LIN {X 0,Y 572.959,Z 555.811,A -85,B 0,C 180,E1 -2247.189,E2 -2247.189} C_VEL
LIN {X 0,Y 572.946,Z 558.187,A -85,B 0,C 180,E1 -2248.595,E2 -2248.595} C_VEL
LIN {X 0,Y 572.938,Z 559,A -85,B 0,C 180,E1 -2250.001,E2 -2250.001} C_VEL
LIN {X 0,Y 572.946,Z 558.185,A -85,B 0,C 180,E1 -2251.407,E2 -2251.407} C_VEL
LIN {X 0,Y 572.938,Z 557.198,A -85,B 0,C 180,E1 -2252.11,E2 -2252.11} C_VEL
LIN {X 0,Y 572.959,Z 555.807,A -85,B 0,C 180,E1 -2252.813,E2 -2252.813} C_VEL
LIN {X 0,Y 573.014,Z 552.893,A -85,B 0,C 180,E1 -2253.869,E2 -2253.869} C_VEL
LIN {X 0,Y 572.963,Z 548.945,A -85,B 0,C 180,E1 -2254.927,E2 -2254.927} C_VEL
LIN {X 0,Y 573.068,Z 542.871,A -85,B 0,C 180,E1 -2256.161,E2 -2256.161} C_VEL
LIN {X 0,Y 573.12,Z 536.231,A -85,B 0,C 180,E1 -2257.222,E2 -2257.222} C_VEL
LIN {X 0,Y 573.193,Z 527.983,A -85,B 0,C 180,E1 -2258.284,E2 -2258.284} C_VEL
LIN {X 0,Y 573.32,Z 517.591,A -85,B 0,C 180,E1 -2259.349,E2 -2259.349} C_VEL
LIN {X 0,Y 573.439,Z 507.912,A -85,B 0,C 180,E1 -2260.148,E2 -2260.148} C_VEL
LIN {X 0,Y 573.55,Z 497.389,A -85,B 0,C 180,E1 -2260.855,E2 -2260.855} C_VEL
LIN {X 0,Y 573.651,Z 485.098,A -85,B 0,C 180,E1 -2261.501,E2 -2261.501} C_VEL
LIN {X 0,Y 573.726,Z 473.144,A -85,B 0,C 180,E1 -2261.976,E2 -2261.976} C_VEL
LIN {X 0,Y 573.815,Z 460.48,A -85,B 0,C 180,E1 -2262.333,E2 -2262.333} C_VEL
LIN {X 0,Y 573.91,Z 447.236,A -85,B 0,C 180,E1 -2262.555,E2 -2262.555} C_VEL
LIN {X 0,Y 573.954,Z 350.648,A -85,B 0,C 180,E1 -2263.77,E2 -2263.77} C_VEL
LIN {X 0,Y 573.391,Z 346.606,A -85,B 0,C 180,E1 -2263.852,E2 -2263.852} C_VEL
LIN {X 0,Y 573.57,Z 326.115,A -85,B 0,C 180,E1 -2266.728,E2 -2266.728} C_VEL
LIN {X 0,Y 573.806,Z 305.604,A -85,B 0,C 180,E1 -2269.647,E2 -2269.647} C_VEL
LIN {X 0,Y 574.032,Z 285.767,A -85,B 0,C 180,E1 -2272.496,E2 -2272.496} C_VEL
LIN {X 0,Y 573.584,Z 280.83,A -85,B 0,C 180,E1 -2273.225,E2 -2273.225} C_VEL
LIN {X 0,Y 573.243,Z 279.083,A -85,B 0,C 180,E1 -2273.497,E2 -2273.497} C_VEL
LIN {X 0,Y 573.263,Z 279.079,A -85,B 0,C 180,E1 -2276.191,E2 -2276.191} C_VEL
LIN {X 0,Y 573.238,Z 279.077,A -85,B 0,C 180,E1 -2278.565,E2 -2278.565} C_VEL
LIN {X 0,Y 573.23,Z 279.074,A -85,B 0,C 180,E1 -2280.994,E2 -2280.994} C_VEL
LIN {X 0,Y 573.247,Z 279.073,A -85,B 0,C 180,E1 -2283.521,E2 -2283.521} C_VEL
LIN {X 0,Y 573.219,Z 279.081,A -85,B 0,C 180,E1 -2286.052,E2 -2286.052} C_VEL
LIN {X 0,Y 573.241,Z 279.079,A -85,B 0,C 180,E1 -2288.702,E2 -2288.702} C_VEL
LIN {X 0,Y 573.233,Z 279.074,A -85,B 0,C 180,E1 -2291.593,E2 -2291.593} C_VEL
LIN {X 0,Y 573.227,Z 279.081,A -85,B 0,C 180,E1 -2294.335,E2 -2294.335} C_VEL
LIN {X 0,Y 573.246,Z 279.073,A -85,B 0,C 180,E1 -2297.359,E2 -2297.359} C_VEL
LIN {X 0,Y 573.242,Z 279.077,A -85,B 0,C 180,E1 -2300.392,E2 -2300.392} C_VEL
LIN {X 0,Y 573.257,Z 279.078,A -85,B 0,C 180,E1 -2303.078,E2 -2303.078} C_VEL
LIN {X 0,Y 573.26,Z 279.071,A -85,B 0,C 180,E1 -2305.671,E2 -2305.671} C_VEL
LIN {X 0,Y 573.243,Z 279.073,A -85,B 0,C 180,E1 -2308.184,E2 -2308.184} C_VEL
LIN {X 0,Y 573.268,Z 279.072,A -85,B 0,C 180,E1 -2310.634,E2 -2310.634} C_VEL
LIN {X 0,Y 573.24,Z 279.079,A -85,B 0,C 180,E1 -2313.508,E2 -2313.508} C_VEL
LIN {X 0,Y 573.228,Z 279.075,A -85,B 0,C 180,E1 -2316.134,E2 -2316.134} C_VEL
LIN {X 0,Y 573.255,Z 279.078,A -85,B 0,C 180,E1 -2319.174,E2 -2319.174} C_VEL
LIN {X 0,Y 573.224,Z 279.085,A -85,B 0,C 180,E1 -2321.411,E2 -2321.411} C_VEL
LIN {X 0,Y 573.247,Z 279.082,A -85,B 0,C 180,E1 -2323.621,E2 -2323.621} C_VEL
LIN {X 0,Y 573.276,Z 279.076,A -85,B 0,C 180,E1 -2325.807,E2 -2325.807} C_VEL
LIN {X 0,Y 573.268,Z 279.069,A -85,B 0,C 180,E1 -2328.745,E2 -2328.745} C_VEL
LIN {X 0,Y 573.258,Z 279.077,A -85,B 0,C 180,E1 -2331.54,E2 -2331.54} C_VEL
LIN {X 0,Y 573.29,Z 279.07,A -85,B 0,C 180,E1 -2334.372,E2 -2334.372} C_VEL
LIN {X 0,Y 573.315,Z 279.072,A -85,B 0,C 180,E1 -2337.892,E2 -2337.892} C_VEL
LIN {X 0,Y 573.332,Z 279.063,A -85,B 0,C 180,E1 -2340.702,E2 -2340.702} C_VEL
LIN {X 0,Y 573.234,Z 279.075,A -85,B 0,C 180,E1 -2343.514,E2 -2343.514} C_VEL
LIN {X 0,Y 573.288,Z 279.068,A -85,B 0,C 180,E1 -2345.628,E2 -2345.628} C_VEL
LIN {X 0,Y 573.274,Z 279.07,A -85,B 0,C 180,E1 -2347.75,E2 -2347.75} C_VEL
LIN {X 0,Y 573.267,Z 279.078,A -85,B 0,C 180,E1 -2350.596,E2 -2350.596} C_VEL
LIN {X 0,Y 573.264,Z 279.077,A -85,B 0,C 180,E1 -2352.748,E2 -2352.748} C_VEL
LIN {X 0,Y 573.237,Z 279.079,A -85,B 0,C 180,E1 -2354.92,E2 -2354.92} C_VEL
LIN {X 0,Y 573.242,Z 279.073,A -85,B 0,C 180,E1 -2357.848,E2 -2357.848} C_VEL
LIN {X 0,Y 573.243,Z 279.074,A -85,B 0,C 180,E1 -2360.077,E2 -2360.077} C_VEL
LIN {X 0,Y 573.235,Z 279.076,A -85,B 0,C 180,E1 -2362.338,E2 -2362.338} C_VEL
LIN {X 0,Y 573.25,Z 279.074,A -85,B 0,C 180,E1 -2364.382,E2 -2364.382} C_VEL
LIN {X 0,Y 572.626,Z 279.16,A -85,B 0,C 180,E1 -2364.968,E2 -2364.968} C_VEL
LIN {X 0,Y 569.786,Z 279.516,A -85,B 0,C 180,E1 -2365.92,E2 -2365.92} C_VEL
LIN {X 0,Y 567.352,Z 279.817,A -85,B 0,C 180,E1 -2366.685,E2 -2366.685} C_VEL
LIN {X 0,Y 566.297,Z 279.944,A -85,B 0,C 180,E1 -2367.277,E2 -2367.277} C_VEL
LIN {X 0,Y 566.207,Z 279.952,A -85,B 0,C 180,E1 -2367.477,E2 -2367.477} C_VEL
LIN {X 0,Y 566.205,Z 279.95,A -85,B 0,C 180,E1 -2369.769,E2 -2369.769} C_VEL
LIN {X 0,Y 566.205,Z 279.95,A -85,B 0,C 180,E1 -2372.429,E2 -2372.429} C_VEL
LIN {X 0,Y 566.182,Z 279.958,A -85,B 0,C 180,E1 -2374.989,E2 -2374.989} C_VEL
LIN {X 0,Y 566.195,Z 279.959,A -85,B 0,C 180,E1 -2377.461,E2 -2377.461} C_VEL
LIN {X 0,Y 566.21,Z 279.949,A -85,B 0,C 180,E1 -2380.199,E2 -2380.199} C_VEL
LIN {X 0,Y 566.203,Z 279.953,A -85,B 0,C 180,E1 -2383.054,E2 -2383.054} C_VEL
LIN {X 0,Y 566.197,Z 279.954,A -85,B 0,C 180,E1 -2386.049,E2 -2386.049} C_VEL
LIN {X 0,Y 566.207,Z 279.952,A -85,B 0,C 180,E1 -2389.214,E2 -2389.214} C_VEL
LIN {X 0,Y 566.186,Z 279.96,A -85,B 0,C 180,E1 -2391.636,E2 -2391.636} C_VEL
LIN {X 0,Y 566.165,Z 279.958,A -85,B 0,C 180,E1 -2394.307,E2 -2394.307} C_VEL
LIN {X 0,Y 566.223,Z 279.947,A -85,B 0,C 180,E1 -2396.897,E2 -2396.897} C_VEL
LIN {X 0,Y 566.183,Z 279.953,A -85,B 0,C 180,E1 -2399.407,E2 -2399.407} C_VEL
LIN {X 0,Y 566.215,Z 279.954,A -85,B 0,C 180,E1 -2401.857,E2 -2401.857} C_VEL
LIN {X 0,Y 566.217,Z 279.958,A -85,B 0,C 180,E1 -2404.25,E2 -2404.25} C_VEL
LIN {X 0,Y 566.175,Z 279.957,A -85,B 0,C 180,E1 -2406.718,E2 -2406.718} C_VEL
LIN {X 0,Y 566.215,Z 279.949,A -85,B 0,C 180,E1 -2409.662,E2 -2409.662} C_VEL
LIN {X 0,Y 566.201,Z 279.957,A -85,B 0,C 180,E1 -2412.668,E2 -2412.668} C_VEL
LIN {X 0,Y 566.231,Z 279.946,A -85,B 0,C 180,E1 -2415.626,E2 -2415.626} C_VEL
LIN {X 0,Y 566.237,Z 279.956,A -85,B 0,C 180,E1 -2418.674,E2 -2418.674} C_VEL
LIN {X 0,Y 566.209,Z 279.951,A -85,B 0,C 180,E1 -2421.433,E2 -2421.433} C_VEL
LIN {X 0,Y 566.256,Z 279.947,A -85,B 0,C 180,E1 -2424.301,E2 -2424.301} C_VEL
LIN {X 0,Y 566.218,Z 279.972,A -85,B 0,C 180,E1 -2425.862,E2 -2425.862} C_VEL
LIN {X 0,Y 566.535,Z 283.112,A -85,B 0,C 180,E1 -2426.443,E2 -2426.443} C_VEL
LIN {X 0,Y 566.304,Z 298.68,A -85,B 0,C 180,E1 -2429.288,E2 -2429.288} C_VEL
LIN {X 0,Y 566.19,Z 308.368,A -85,B 0,C 180,E1 -2431.044,E2 -2431.044} C_VEL
LIN {X 0,Y 567.18,Z 314.204,A -85,B 0,C 180,E1 -2431.153,E2 -2431.153} C_VEL
LIN {X 0,Y 566.873,Z 414.703,A -85,B 0,C 180,E1 -2432.441,E2 -2432.441} C_VEL
LIN {X 0,Y 566.763,Z 427.913,A -85,B 0,C 180,E1 -2432.753,E2 -2432.753} C_VEL
LIN {X 0,Y 566.723,Z 440.499,A -85,B 0,C 180,E1 -2433.198,E2 -2433.198} C_VEL
LIN {X 0,Y 566.588,Z 451.79,A -85,B 0,C 180,E1 -2433.733,E2 -2433.733} C_VEL
LIN {X 0,Y 566.408,Z 463.445,A -85,B 0,C 180,E1 -2434.447,E2 -2434.447} C_VEL
LIN {X 0,Y 566.309,Z 473.897,A -85,B 0,C 180,E1 -2435.25,E2 -2435.25} C_VEL
LIN {X 0,Y 566.171,Z 482.489,A -85,B 0,C 180,E1 -2436.056,E2 -2436.056} C_VEL
LIN {X 0,Y 566.111,Z 490.229,A -85,B 0,C 180,E1 -2436.928,E2 -2436.928} C_VEL
LIN {X 0,Y 566.043,Z 498.223,A -85,B 0,C 180,E1 -2438.028,E2 -2438.028} C_VEL
LIN {X 0,Y 565.981,Z 503.555,A -85,B 0,C 180,E1 -2438.928,E2 -2438.928} C_VEL
LIN {X 0,Y 565.946,Z 508.754,A -85,B 0,C 180,E1 -2440.011,E2 -2440.011} C_VEL
LIN {X 0,Y 565.929,Z 513.016,A -85,B 0,C 180,E1 -2441.169,E2 -2441.169} C_VEL
LIN {X 0,Y 565.867,Z 515.788,A -85,B 0,C 180,E1 -2442.188,E2 -2442.188} C_VEL
LIN {X 0,Y 565.843,Z 517.211,A -85,B 0,C 180,E1 -2442.917,E2 -2442.917} C_VEL
LIN {X 0,Y 565.861,Z 518.215,A -85,B 0,C 180,E1 -2443.648,E2 -2443.648} C_VEL
LIN {X 0,Y 565.873,Z 518.817,A -85,B 0,C 180,E1 -2444.381,E2 -2444.381} C_VEL
LIN {X 0,Y 565.803,Z 518.99,A -85,B 0,C 180,E1 -2445.119,E2 -2445.119} C_VEL
LIN {X 0,Y 565.81,Z 518.719,A -85,B 0,C 180,E1 -2445.857,E2 -2445.857} C_VEL
LIN {X 0,Y 565.851,Z 517.497,A -85,B 0,C 180,E1 -2446.99,E2 -2446.99} C_VEL
LIN {X 0,Y 565.892,Z 514.38,A -85,B 0,C 180,E1 -2448.462,E2 -2448.462} C_VEL
LIN {X 0,Y 565.926,Z 510.712,A -85,B 0,C 180,E1 -2449.59,E2 -2449.59} C_VEL
LIN {X 0,Y 565.944,Z 505.785,A -85,B 0,C 180,E1 -2450.726,E2 -2450.726} C_VEL
LIN {X 0,Y 566.004,Z 499.43,A -85,B 0,C 180,E1 -2451.869,E2 -2451.869} C_VEL
LIN {X 0,Y 566.077,Z 491.551,A -85,B 0,C 180,E1 -2452.998,E2 -2452.998} C_VEL
LIN {X 0,Y 566.184,Z 482.955,A -85,B 0,C 180,E1 -2453.985,E2 -2453.985} C_VEL
LIN {X 0,Y 566.315,Z 473.683,A -85,B 0,C 180,E1 -2454.858,E2 -2454.858} C_VEL
LIN {X 0,Y 566.454,Z 463.473,A -85,B 0,C 180,E1 -2455.64,E2 -2455.64} C_VEL
LIN {X 0,Y 566.6,Z 452.432,A -85,B 0,C 180,E1 -2456.322,E2 -2456.322} C_VEL
LIN {X 0,Y 566.745,Z 440.606,A -85,B 0,C 180,E1 -2456.888,E2 -2456.888} C_VEL
LIN {X 0,Y 566.832,Z 428.098,A -85,B 0,C 180,E1 -2457.33,E2 -2457.33} C_VEL
LIN {X 0,Y 566.919,Z 414.525,A -85,B 0,C 180,E1 -2457.651,E2 -2457.651} C_VEL
LIN {X 0,Y 567.043,Z 313.459,A -85,B 0,C 180,E1 -2458.95,E2 -2458.95} C_VEL
LIN {X 0,Y 566.206,Z 308.331,A -85,B 0,C 180,E1 -2459.053,E2 -2459.053} C_VEL
LIN {X 0,Y 566.364,Z 293.061,A -85,B 0,C 180,E1 -2461.827,E2 -2461.827} C_VEL
LIN {X 0,Y 566.379,Z 281.442,A -85,B 0,C 180,E1 -2463.943,E2 -2463.943} C_VEL
LIN {X 0,Y 566.14,Z 279.963,A -85,B 0,C 180,E1 -2464.227,E2 -2464.227} C_VEL
LIN {X 0,Y 566.176,Z 279.962,A -85,B 0,C 180,E1 -2467.461,E2 -2467.461} C_VEL
LIN {X 0,Y 566.181,Z 279.954,A -85,B 0,C 180,E1 -2470.199,E2 -2470.199} C_VEL
LIN {X 0,Y 566.13,Z 279.965,A -85,B 0,C 180,E1 -2473.059,E2 -2473.059} C_VEL
LIN {X 0,Y 566.143,Z 279.958,A -85,B 0,C 180,E1 -2476.052,E2 -2476.052} C_VEL
LIN {X 0,Y 566.142,Z 279.959,A -85,B 0,C 180,E1 -2478.858,E2 -2478.858} C_VEL
LIN {X 0,Y 566.186,Z 279.961,A -85,B 0,C 180,E1 -2481.442,E2 -2481.442} C_VEL
LIN {X 0,Y 566.125,Z 279.958,A -85,B 0,C 180,E1 -2484.305,E2 -2484.305} C_VEL
LIN {X 0,Y 566.189,Z 279.953,A -85,B 0,C 180,E1 -2486.896,E2 -2486.896} C_VEL
LIN {X 0,Y 566.162,Z 279.959,A -85,B 0,C 180,E1 -2489.406,E2 -2489.406} C_VEL
LIN {X 0,Y 566.172,Z 279.964,A -85,B 0,C 180,E1 -2491.855,E2 -2491.855} C_VEL
LIN {X 0,Y 566.222,Z 279.947,A -85,B 0,C 180,E1 -2495.039,E2 -2495.039} C_VEL
LIN {X 0,Y 566.176,Z 279.96,A -85,B 0,C 180,E1 -2498.137,E2 -2498.137} C_VEL
LIN {X 0,Y 566.215,Z 279.951,A -85,B 0,C 180,E1 -2500.613,E2 -2500.613} C_VEL
LIN {X 0,Y 566.163,Z 279.955,A -85,B 0,C 180,E1 -2503.411,E2 -2503.411} C_VEL
LIN {X 0,Y 566.174,Z 279.96,A -85,B 0,C 180,E1 -2506.358,E2 -2506.358} C_VEL
LIN {X 0,Y 566.219,Z 279.951,A -85,B 0,C 180,E1 -2508.675,E2 -2508.675} C_VEL
LIN {X 0,Y 566.21,Z 279.949,A -85,B 0,C 180,E1 -2511.434,E2 -2511.434} C_VEL
LIN {X 0,Y 566.243,Z 279.953,A -85,B 0,C 180,E1 -2514.302,E2 -2514.302} C_VEL
LIN {X 0,Y 566.256,Z 279.944,A -85,B 0,C 180,E1 -2517.866,E2 -2517.866} C_VEL
LIN {X 0,Y 566.297,Z 279.945,A -85,B 0,C 180,E1 -2520.711,E2 -2520.711} C_VEL
LIN {X 0,Y 566.173,Z 279.952,A -85,B 0,C 180,E1 -2523.559,E2 -2523.559} C_VEL
LIN {X 0,Y 566.243,Z 279.945,A -85,B 0,C 180,E1 -2525.699,E2 -2525.699} C_VEL
LIN {X 0,Y 566.22,Z 279.955,A -85,B 0,C 180,E1 -2528.566,E2 -2528.566} C_VEL
LIN {X 0,Y 566.237,Z 279.947,A -85,B 0,C 180,E1 -2531.455,E2 -2531.455} C_VEL
LIN {X 0,Y 566.22,Z 279.951,A -85,B 0,C 180,E1 -2534.507,E2 -2534.507} C_VEL
LIN {X 0,Y 566.186,Z 279.955,A -85,B 0,C 180,E1 -2537.332,E2 -2537.332} C_VEL
LIN {X 0,Y 566.2,Z 279.951,A -85,B 0,C 180,E1 -2540.338,E2 -2540.338} C_VEL
LIN {X 0,Y 566.177,Z 279.957,A -85,B 0,C 180,E1 -2543.405,E2 -2543.405} C_VEL
LIN {X 0,Y 566.215,Z 279.95,A -85,B 0,C 180,E1 -2545.749,E2 -2545.749} C_VEL
LIN {X 0,Y 566.19,Z 279.95,A -85,B 0,C 180,E1 -2548.203,E2 -2548.203} C_VEL
LIN {X 0,Y 566.183,Z 279.954,A -85,B 0,C 180,E1 -2550.593,E2 -2550.593} C_VEL
LIN {X 0,Y 566.218,Z 279.954,A -85,B 0,C 180,E1 -2553.103,E2 -2553.103} C_VEL
LIN {X 0,Y 566.202,Z 279.955,A -85,B 0,C 180,E1 -2555.69,E2 -2555.69} C_VEL
LIN {X 0,Y 566.207,Z 279.95,A -85,B 0,C 180,E1 -2558.56,E2 -2558.56} C_VEL
LIN {X 0,Y 566.203,Z 279.955,A -85,B 0,C 180,E1 -2561.137,E2 -2561.137} C_VEL
LIN {X 0,Y 566.192,Z 279.954,A -85,B 0,C 180,E1 -2564.037,E2 -2564.037} C_VEL
LIN {X 0,Y 566.198,Z 279.952,A -85,B 0,C 180,E1 -2567.084,E2 -2567.084} C_VEL
LIN {X 0,Y 566.22,Z 279.956,A -85,B 0,C 180,E1 -2569.804,E2 -2569.804} C_VEL
LIN {X 0,Y 566.194,Z 279.952,A -85,B 0,C 180,E1 -2572.6,E2 -2572.6} C_VEL
LIN {X 0,Y 566.204,Z 279.952,A -85,B 0,C 180,E1 -2575.184,E2 -2575.184} C_VEL
LIN {X 0,Y 566.226,Z 279.956,A -85,B 0,C 180,E1 -2577.745,E2 -2577.745} C_VEL
LIN {X 0,Y 566.2,Z 279.956,A -85,B 0,C 180,E1 -2580.329,E2 -2580.329} C_VEL
LIN {X 0,Y 566.216,Z 279.951,A -85,B 0,C 180,E1 -2582.663,E2 -2582.663} C_VEL
LIN {X 0,Y 566.234,Z 279.949,A -85,B 0,C 180,E1 -2585.04,E2 -2585.04} C_VEL
LIN {X 0,Y 566.222,Z 280.105,A -85,B 0,C 180,E1 -2586.405,E2 -2586.405} C_VEL
LIN {X 0,Y 567.058,Z 285.451,A -85,B 0,C 180,E1 -2587.214,E2 -2587.214} C_VEL
LIN {X 0,Y 566.867,Z 306.727,A -85,B 0,C 180,E1 -2590.275,E2 -2590.275} C_VEL
LIN {X 0,Y 566.598,Z 327.558,A -85,B 0,C 180,E1 -2593.267,E2 -2593.267} C_VEL
LIN {X 0,Y 566.392,Z 346.703,A -85,B 0,C 180,E1 -2595.987,E2 -2595.987} C_VEL
LIN {X 0,Y 567.202,Z 353.339,A -85,B 0,C 180,E1 -2596.097,E2 -2596.097} C_VEL
LIN {X 0,Y 566.952,Z 455.008,A -85,B 0,C 180,E1 -2597.404,E2 -2597.404} C_VEL
LIN {X 0,Y 566.836,Z 468.259,A -85,B 0,C 180,E1 -2597.72,E2 -2597.72} C_VEL
LIN {X 0,Y 566.719,Z 480.407,A -85,B 0,C 180,E1 -2598.149,E2 -2598.149} C_VEL
LIN {X 0,Y 566.626,Z 492.089,A -85,B 0,C 180,E1 -2598.705,E2 -2598.705} C_VEL
LIN {X 0,Y 566.487,Z 502.924,A -85,B 0,C 180,E1 -2599.367,E2 -2599.367} C_VEL
LIN {X 0,Y 566.329,Z 513.554,A -85,B 0,C 180,E1 -2600.177,E2 -2600.177} C_VEL
LIN {X 0,Y 566.205,Z 523.094,A -85,B 0,C 180,E1 -2601.075,E2 -2601.075} C_VEL
LIN {X 0,Y 566.11,Z 530.97,A -85,B 0,C 180,E1 -2601.973,E2 -2601.973} C_VEL
LIN {X 0,Y 566.004,Z 538.629,A -85,B 0,C 180,E1 -2603.048,E2 -2603.048} C_VEL
LIN {X 0,Y 566.004,Z 545.685,A -85,B 0,C 180,E1 -2604.3,E2 -2604.3} C_VEL
LIN {X 0,Y 565.933,Z 550.377,A -85,B 0,C 180,E1 -2605.371,E2 -2605.371} C_VEL
LIN {X 0,Y 565.926,Z 553.961,A -85,B 0,C 180,E1 -2606.441,E2 -2606.441} C_VEL
LIN {X 0,Y 565.877,Z 555.81,A -85,B 0,C 180,E1 -2607.154,E2 -2607.154} C_VEL
LIN {X 0,Y 565.845,Z 558.186,A -85,B 0,C 180,E1 -2608.578,E2 -2608.578} C_VEL
LIN {X 0,Y 565.839,Z 559,A -85,B 0,C 180,E1 -2610.001,E2 -2610.001} C_VEL
LIN {X 0,Y 565.845,Z 558.184,A -85,B 0,C 180,E1 -2611.424,E2 -2611.424} C_VEL
LIN {X 0,Y 565.878,Z 555.808,A -85,B 0,C 180,E1 -2612.849,E2 -2612.849} C_VEL
LIN {X 0,Y 565.926,Z 552.893,A -85,B 0,C 180,E1 -2613.917,E2 -2613.917} C_VEL
LIN {X 0,Y 565.878,Z 548.945,A -85,B 0,C 180,E1 -2614.988,E2 -2614.988} C_VEL
LIN {X 0,Y 565.994,Z 542.871,A -85,B 0,C 180,E1 -2616.238,E2 -2616.238} C_VEL
LIN {X 0,Y 566.053,Z 536.23,A -85,B 0,C 180,E1 -2617.312,E2 -2617.312} C_VEL
LIN {X 0,Y 566.142,Z 527.983,A -85,B 0,C 180,E1 -2618.388,E2 -2618.388} C_VEL
LIN {X 0,Y 566.254,Z 519.529,A -85,B 0,C 180,E1 -2619.286,E2 -2619.286} C_VEL
LIN {X 0,Y 566.393,Z 509.083,A -85,B 0,C 180,E1 -2620.185,E2 -2620.185} C_VEL
LIN {X 0,Y 566.571,Z 497.689,A -85,B 0,C 180,E1 -2620.972,E2 -2620.972} C_VEL
LIN {X 0,Y 566.693,Z 485.866,A -85,B 0,C 180,E1 -2621.609,E2 -2621.609} C_VEL
LIN {X 0,Y 566.777,Z 473.142,A -85,B 0,C 180,E1 -2622.125,E2 -2622.125} C_VEL
LIN {X 0,Y 566.878,Z 460.479,A -85,B 0,C 180,E1 -2622.486,E2 -2622.486} C_VEL
LIN {X 0,Y 566.978,Z 447.236,A -85,B 0,C 180,E1 -2622.711,E2 -2622.711} C_VEL
LIN {X 0,Y 567.048,Z 351.206,A -85,B 0,C 180,E1 -2623.934,E2 -2623.934} C_VEL
LIN {X 0,Y 566.385,Z 346.606,A -85,B 0,C 180,E1 -2624.026,E2 -2624.026} C_VEL
LIN {X 0,Y 566.613,Z 324.886,A -85,B 0,C 180,E1 -2627.116,E2 -2627.116} C_VEL
LIN {X 0,Y 566.87,Z 303.955,A -85,B 0,C 180,E1 -2630.124,E2 -2630.124} C_VEL
LIN {X 0,Y 567.057,Z 285.517,A -85,B 0,C 180,E1 -2632.788,E2 -2632.788} C_VEL
LIN {X 0,Y 566.21,Z 279.959,A -85,B 0,C 180,E1 -2633.646,E2 -2633.646} C_VEL
LIN {X 0,Y 566.212,Z 279.958,A -85,B 0,C 180,E1 -2635.75,E2 -2635.75} C_VEL
LIN {X 0,Y 566.209,Z 279.958,A -85,B 0,C 180,E1 -2638.203,E2 -2638.203} C_VEL
LIN {X 0,Y 566.195,Z 279.951,A -85,B 0,C 180,E1 -2641.077,E2 -2641.077} C_VEL
LIN {X 0,Y 566.203,Z 279.952,A -85,B 0,C 180,E1 -2643.732,E2 -2643.732} C_VEL
LIN {X 0,Y 566.205,Z 279.956,A -85,B 0,C 180,E1 -2646.57,E2 -2646.57} C_VEL
LIN {X 0,Y 566.217,Z 279.948,A -85,B 0,C 180,E1 -2649.686,E2 -2649.686} C_VEL
LIN {X 0,Y 566.206,Z 279.954,A -85,B 0,C 180,E1 -2652.917,E2 -2652.917} C_VEL
LIN {X 0,Y 566.199,Z 279.952,A -85,B 0,C 180,E1 -2656.049,E2 -2656.049} C_VEL
LIN {X 0,Y 566.209,Z 279.952,A -85,B 0,C 180,E1 -2659.215,E2 -2659.215} C_VEL
LIN {X 0,Y 566.188,Z 279.952,A -85,B 0,C 180,E1 -2661.637,E2 -2661.637} C_VEL
LIN {X 0,Y 566.167,Z 279.956,A -85,B 0,C 180,E1 -2664.308,E2 -2664.308} C_VEL
LIN {X 0,Y 566.205,Z 279.958,A -85,B 0,C 180,E1 -2666.897,E2 -2666.897} C_VEL
LIN {X 0,Y 566.185,Z 279.957,A -85,B 0,C 180,E1 -2669.407,E2 -2669.407} C_VEL
LIN {X 0,Y 566.199,Z 279.951,A -85,B 0,C 180,E1 -2671.856,E2 -2671.856} C_VEL
LIN {X 0,Y 566.213,Z 279.948,A -85,B 0,C 180,E1 -2674.251,E2 -2674.251} C_VEL
LIN {X 0,Y 566.173,Z 279.955,A -85,B 0,C 180,E1 -2676.72,E2 -2676.72} C_VEL
LIN {X 0,Y 566.212,Z 279.955,A -85,B 0,C 180,E1 -2679.663,E2 -2679.663} C_VEL
LIN {X 0,Y 566.199,Z 279.95,A -85,B 0,C 180,E1 -2682.668,E2 -2682.668} C_VEL
LIN {X 0,Y 566.238,Z 279.956,A -85,B 0,C 180,E1 -2685.627,E2 -2685.627} C_VEL
LIN {X 0,Y 566.24,Z 279.945,A -85,B 0,C 180,E1 -2688.675,E2 -2688.675} C_VEL
LIN {X 0,Y 566.209,Z 279.953,A -85,B 0,C 180,E1 -2691.434,E2 -2691.434} C_VEL
LIN {X 0,Y 566.256,Z 279.947,A -85,B 0,C 180,E1 -2694.302,E2 -2694.302} C_VEL
LIN {X 0,Y 566.286,Z 279.947,A -85,B 0,C 180,E1 -2697.866,E2 -2697.866} C_VEL
LIN {X 0,Y 566.303,Z 279.939,A -85,B 0,C 180,E1 -2700.711,E2 -2700.711} C_VEL
LIN {X 0,Y 566.273,Z 279.942,A -85,B 0,C 180,E1 -2702.845,E2 -2702.845} C_VEL
LIN {X 0,Y 566.256,Z 279.945,A -85,B 0,C 180,E1 -2705.698,E2 -2705.698} C_VEL
LIN {X 0,Y 566.209,Z 279.956,A -85,B 0,C 180,E1 -2708.566,E2 -2708.566} C_VEL
LIN {X 0,Y 566.247,Z 279.944,A -85,B 0,C 180,E1 -2711.454,E2 -2711.454} C_VEL
LIN {X 0,Y 566.234,Z 279.955,A -85,B 0,C 180,E1 -2714.504,E2 -2714.504} C_VEL
LIN {X 0,Y 566.201,Z 279.951,A -85,B 0,C 180,E1 -2717.331,E2 -2717.331} C_VEL
LIN {X 0,Y 566.21,Z 279.952,A -85,B 0,C 180,E1 -2720.337,E2 -2720.337} C_VEL
LIN {X 0,Y 566.172,Z 279.957,A -85,B 0,C 180,E1 -2723.28,E2 -2723.28} C_VEL
LIN {X 0,Y 566.217,Z 279.948,A -85,B 0,C 180,E1 -2725.749,E2 -2725.749} C_VEL
LIN {X 0,Y 566.207,Z 279.952,A -85,B 0,C 180,E1 -2727.477,E2 -2727.477} C_VEL
LIN {X 0,Y 565.527,Z 280.037,A -85,B 0,C 180,E1 -2728.071,E2 -2728.071} C_VEL
LIN {X 0,Y 562.661,Z 280.402,A -85,B 0,C 180,E1 -2729.034,E2 -2729.034} C_VEL
LIN {X 0,Y 560.251,Z 280.696,A -85,B 0,C 180,E1 -2729.81,E2 -2729.81} C_VEL
LIN {X 0,Y 559.223,Z 280.82,A -85,B 0,C 180,E1 -2730.408,E2 -2730.408} C_VEL
LIN {X 0,Y 559.143,Z 280.832,A -85,B 0,C 180,E1 -2730.611,E2 -2730.611} C_VEL
LIN {X 0,Y 559.166,Z 280.831,A -85,B 0,C 180,E1 -2733.575,E2 -2733.575} C_VEL
LIN {X 0,Y 559.133,Z 280.831,A -85,B 0,C 180,E1 -2736.442,E2 -2736.442} C_VEL
LIN {X 0,Y 559.176,Z 280.828,A -85,B 0,C 180,E1 -2738.934,E2 -2738.934} C_VEL
LIN {X 0,Y 559.167,Z 280.832,A -85,B 0,C 180,E1 -2741.77,E2 -2741.77} C_VEL
LIN {X 0,Y 559.135,Z 280.83,A -85,B 0,C 180,E1 -2744.74,E2 -2744.74} C_VEL
LIN {X 0,Y 559.161,Z 280.831,A -85,B 0,C 180,E1 -2747.256,E2 -2747.256} C_VEL
LIN {X 0,Y 559.181,Z 280.829,A -85,B 0,C 180,E1 -2750.134,E2 -2750.134} C_VEL
LIN {X 0,Y 559.144,Z 280.829,A -85,B 0,C 180,E1 -2752.891,E2 -2752.891} C_VEL
LIN {X 0,Y 559.169,Z 280.835,A -85,B 0,C 180,E1 -2756.05,E2 -2756.05} C_VEL
LIN {X 0,Y 559.157,Z 280.827,A -85,B 0,C 180,E1 -2758.98,E2 -2758.98} C_VEL
LIN {X 0,Y 559.172,Z 280.828,A -85,B 0,C 180,E1 -2761.618,E2 -2761.618} C_VEL
LIN {X 0,Y 559.184,Z 280.829,A -85,B 0,C 180,E1 -2763.902,E2 -2763.902} C_VEL
LIN {X 0,Y 559.145,Z 280.835,A -85,B 0,C 180,E1 -2766.57,E2 -2766.57} C_VEL
LIN {X 0,Y 559.182,Z 280.824,A -85,B 0,C 180,E1 -2769.395,E2 -2769.395} C_VEL
LIN {X 0,Y 559.143,Z 280.83,A -85,B 0,C 180,E1 -2771.685,E2 -2771.685} C_VEL
LIN {X 0,Y 559.166,Z 280.828,A -85,B 0,C 180,E1 -2773.947,E2 -2773.947} C_VEL
LIN {X 0,Y 559.17,Z 280.829,A -85,B 0,C 180,E1 -2776.183,E2 -2776.183} C_VEL
LIN {X 0,Y 559.208,Z 280.83,A -85,B 0,C 180,E1 -2778.604,E2 -2778.604} C_VEL
LIN {X 0,Y 559.173,Z 280.829,A -85,B 0,C 180,E1 -2781.324,E2 -2781.324} C_VEL
LIN {X 0,Y 559.225,Z 280.823,A -85,B 0,C 180,E1 -2784.229,E2 -2784.229} C_VEL
LIN {X 0,Y 559.18,Z 280.84,A -85,B 0,C 180,E1 -2785.81,E2 -2785.81} C_VEL
LIN {X 0,Y 559.473,Z 285.017,A -85,B 0,C 180,E1 -2786.578,E2 -2786.578} C_VEL
LIN {X 0,Y 559.277,Z 299.735,A -85,B 0,C 180,E1 -2789.279,E2 -2789.279} C_VEL
LIN {X 0,Y 559.173,Z 308.573,A -85,B 0,C 180,E1 -2790.877,E2 -2790.877} C_VEL
LIN {X 0,Y 560.267,Z 314.934,A -85,B 0,C 180,E1 -2790.987,E2 -2790.987} C_VEL
LIN {X 0,Y 559.941,Z 415.154,A -85,B 0,C 180,E1 -2792.292,E2 -2792.292} C_VEL
LIN {X 0,Y 559.827,Z 428.204,A -85,B 0,C 180,E1 -2792.607,E2 -2792.607} C_VEL
LIN {X 0,Y 559.776,Z 440.715,A -85,B 0,C 180,E1 -2793.058,E2 -2793.058} C_VEL
LIN {X 0,Y 559.619,Z 451.958,A -85,B 0,C 180,E1 -2793.599,E2 -2793.599} C_VEL
LIN {X 0,Y 559.408,Z 463.576,A -85,B 0,C 180,E1 -2794.322,E2 -2794.322} C_VEL
LIN {X 0,Y 559.31,Z 474,A -85,B 0,C 180,E1 -2795.135,E2 -2795.135} C_VEL
LIN {X 0,Y 559.12,Z 482.587,A -85,B 0,C 180,E1 -2795.951,E2 -2795.951} C_VEL
LIN {X 0,Y 559.069,Z 490.681,A -85,B 0,C 180,E1 -2796.88,E2 -2796.88} C_VEL
LIN {X 0,Y 558.98,Z 498.281,A -85,B 0,C 180,E1 -2797.948,E2 -2797.948} C_VEL
LIN {X 0,Y 558.877,Z 504.538,A -85,B 0,C 180,E1 -2799.043,E2 -2799.043} C_VEL
LIN {X 0,Y 558.852,Z 509.517,A -85,B 0,C 180,E1 -2800.139,E2 -2800.139} C_VEL
LIN {X 0,Y 558.844,Z 513.281,A -85,B 0,C 180,E1 -2801.209,E2 -2801.209} C_VEL
LIN {X 0,Y 558.772,Z 516.187,A -85,B 0,C 180,E1 -2802.345,E2 -2802.345} C_VEL
LIN {X 0,Y 558.742,Z 517.512,A -85,B 0,C 180,E1 -2803.084,E2 -2803.084} C_VEL
LIN {X 0,Y 558.786,Z 518.854,A -85,B 0,C 180,E1 -2804.431,E2 -2804.431} C_VEL
LIN {X 0,Y 558.706,Z 518.947,A -85,B 0,C 180,E1 -2805.316,E2 -2805.316} C_VEL
LIN {X 0,Y 558.727,Z 518.588,A -85,B 0,C 180,E1 -2806.064,E2 -2806.064} C_VEL
LIN {X 0,Y 558.76,Z 517.4,A -85,B 0,C 180,E1 -2807.076,E2 -2807.076} C_VEL
LIN {X 0,Y 558.777,Z 514.835,A -85,B 0,C 180,E1 -2808.325,E2 -2808.325} C_VEL
LIN {X 0,Y 558.826,Z 511.585,A -85,B 0,C 180,E1 -2809.399,E2 -2809.399} C_VEL
LIN {X 0,Y 558.841,Z 506.657,A -85,B 0,C 180,E1 -2810.616,E2 -2810.616} C_VEL
LIN {X 0,Y 558.913,Z 500.718,A -85,B 0,C 180,E1 -2811.746,E2 -2811.746} C_VEL
LIN {X 0,Y 559.001,Z 492.76,A -85,B 0,C 180,E1 -2812.937,E2 -2812.937} C_VEL
LIN {X 0,Y 559.134,Z 484.696,A -85,B 0,C 180,E1 -2813.912,E2 -2813.912} C_VEL
LIN {X 0,Y 559.292,Z 474.717,A -85,B 0,C 180,E1 -2814.894,E2 -2814.894} C_VEL
LIN {X 0,Y 559.458,Z 463.372,A -85,B 0,C 180,E1 -2815.782,E2 -2815.782} C_VEL
LIN {X 0,Y 559.629,Z 452.253,A -85,B 0,C 180,E1 -2816.474,E2 -2816.474} C_VEL
LIN {X 0,Y 559.806,Z 440.738,A -85,B 0,C 180,E1 -2817.031,E2 -2817.031} C_VEL
LIN {X 0,Y 559.898,Z 428.358,A -85,B 0,C 180,E1 -2817.477,E2 -2817.477} C_VEL
LIN {X 0,Y 559.982,Z 415.296,A -85,B 0,C 180,E1 -2817.794,E2 -2817.794} C_VEL
LIN {X 0,Y 560.224,Z 314.878,A -85,B 0,C 180,E1 -2819.105,E2 -2819.105} C_VEL
LIN {X 0,Y 559.186,Z 308.391,A -85,B 0,C 180,E1 -2819.221,E2 -2819.221} C_VEL
LIN {X 0,Y 559.346,Z 292.939,A -85,B 0,C 180,E1 -2822.054,E2 -2822.054} C_VEL
LIN {X 0,Y 559.328,Z 282.22,A -85,B 0,C 180,E1 -2823.974,E2 -2823.974} C_VEL
LIN {X 0,Y 559.104,Z 280.84,A -85,B 0,C 180,E1 -2824.25,E2 -2824.25} C_VEL
LIN {X 0,Y 559.105,Z 280.844,A -85,B 0,C 180,E1 -2827.109,E2 -2827.109} C_VEL
LIN {X 0,Y 559.133,Z 280.833,A -85,B 0,C 180,E1 -2829.938,E2 -2829.938} C_VEL
LIN {X 0,Y 559.097,Z 280.838,A -85,B 0,C 180,E1 -2832.747,E2 -2832.747} C_VEL
LIN {X 0,Y 559.109,Z 280.838,A -85,B 0,C 180,E1 -2835.763,E2 -2835.763} C_VEL
LIN {X 0,Y 559.111,Z 280.835,A -85,B 0,C 180,E1 -2838.225,E2 -2838.225} C_VEL
LIN {X 0,Y 559.154,Z 280.833,A -85,B 0,C 180,E1 -2841.192,E2 -2841.192} C_VEL
LIN {X 0,Y 559.1,Z 280.839,A -85,B 0,C 180,E1 -2843.786,E2 -2843.786} C_VEL
LIN {X 0,Y 559.133,Z 280.832,A -85,B 0,C 180,E1 -2846.423,E2 -2846.423} C_VEL
LIN {X 0,Y 559.138,Z 280.83,A -85,B 0,C 180,E1 -2848.98,E2 -2848.98} C_VEL
LIN {X 0,Y 559.119,Z 280.84,A -85,B 0,C 180,E1 -2851.625,E2 -2851.625} C_VEL
LIN {X 0,Y 559.164,Z 280.826,A -85,B 0,C 180,E1 -2854.813,E2 -2854.813} C_VEL
LIN {X 0,Y 559.124,Z 280.841,A -85,B 0,C 180,E1 -2857.847,E2 -2857.847} C_VEL
LIN {X 0,Y 559.176,Z 280.829,A -85,B 0,C 180,E1 -2860.494,E2 -2860.494} C_VEL
LIN {X 0,Y 559.141,Z 280.828,A -85,B 0,C 180,E1 -2863.196,E2 -2863.196} C_VEL
LIN {X 0,Y 559.148,Z 280.839,A -85,B 0,C 180,E1 -2866.184,E2 -2866.184} C_VEL
LIN {X 0,Y 559.19,Z 280.827,A -85,B 0,C 180,E1 -2868.605,E2 -2868.605} C_VEL
LIN {X 0,Y 559.169,Z 280.826,A -85,B 0,C 180,E1 -2871.325,E2 -2871.325} C_VEL
LIN {X 0,Y 559.21,Z 280.828,A -85,B 0,C 180,E1 -2874.23,E2 -2874.23} C_VEL
LIN {X 0,Y 559.228,Z 280.819,A -85,B 0,C 180,E1 -2877.839,E2 -2877.839} C_VEL
LIN {X 0,Y 559.266,Z 280.821,A -85,B 0,C 180,E1 -2880.72,E2 -2880.72} C_VEL
LIN {X 0,Y 559.234,Z 280.821,A -85,B 0,C 180,E1 -2882.882,E2 -2882.882} C_VEL
LIN {X 0,Y 559.212,Z 280.821,A -85,B 0,C 180,E1 -2885.771,E2 -2885.771} C_VEL
LIN {X 0,Y 559.179,Z 280.833,A -85,B 0,C 180,E1 -2888.675,E2 -2888.675} C_VEL
LIN {X 0,Y 559.195,Z 280.823,A -85,B 0,C 180,E1 -2891.601,E2 -2891.601} C_VEL
LIN {X 0,Y 559.186,Z 280.828,A -85,B 0,C 180,E1 -2894.596,E2 -2894.596} C_VEL
LIN {X 0,Y 559.146,Z 280.83,A -85,B 0,C 180,E1 -2897.558,E2 -2897.558} C_VEL
LIN {X 0,Y 559.159,Z 280.827,A -85,B 0,C 180,E1 -2899.838,E2 -2899.838} C_VEL
LIN {X 0,Y 559.128,Z 280.831,A -85,B 0,C 180,E1 -2902.154,E2 -2902.154} C_VEL
LIN {X 0,Y 559.167,Z 280.836,A -85,B 0,C 180,E1 -2905.188,E2 -2905.188} C_VEL
LIN {X 0,Y 559.181,Z 280.825,A -85,B 0,C 180,E1 -2907.712,E2 -2907.712} C_VEL
LIN {X 0,Y 559.158,Z 280.828,A -85,B 0,C 180,E1 -2910.183,E2 -2910.183} C_VEL
LIN {X 0,Y 559.165,Z 280.828,A -85,B 0,C 180,E1 -2912.715,E2 -2912.715} C_VEL
LIN {X 0,Y 559.147,Z 280.839,A -85,B 0,C 180,E1 -2915.323,E2 -2915.323} C_VEL
LIN {X 0,Y 559.126,Z 280.834,A -85,B 0,C 180,E1 -2918.018,E2 -2918.018} C_VEL
LIN {X 0,Y 559.168,Z 280.828,A -85,B 0,C 180,E1 -2920.812,E2 -2920.812} C_VEL
LIN {X 0,Y 559.154,Z 280.835,A -85,B 0,C 180,E1 -2923.733,E2 -2923.733} C_VEL
LIN {X 0,Y 559.161,Z 280.826,A -85,B 0,C 180,E1 -2926.802,E2 -2926.802} C_VEL
LIN {X 0,Y 559.17,Z 280.829,A -85,B 0,C 180,E1 -2929.191,E2 -2929.191} C_VEL
LIN {X 0,Y 559.129,Z 280.838,A -85,B 0,C 180,E1 -2931.984,E2 -2931.984} C_VEL
LIN {X 0,Y 559.14,Z 280.831,A -85,B 0,C 180,E1 -2934.679,E2 -2934.679} C_VEL
LIN {X 0,Y 559.151,Z 280.831,A -85,B 0,C 180,E1 -2937.366,E2 -2937.366} C_VEL
LIN {X 0,Y 559.145,Z 280.837,A -85,B 0,C 180,E1 -2940.144,E2 -2940.144} C_VEL
LIN {X 0,Y 559.168,Z 280.829,A -85,B 0,C 180,E1 -2943.099,E2 -2943.099} C_VEL
LIN {X 0,Y 559.18,Z 280.836,A -85,B 0,C 180,E1 -2946.09,E2 -2946.09} C_VEL
LIN {X 0,Y 559.18,Z 280.949,A -85,B 0,C 180,E1 -2946.262,E2 -2946.262} C_VEL
LIN {X 0,Y 560.097,Z 286.465,A -85,B 0,C 180,E1 -2947.11,E2 -2947.11} C_VEL
LIN {X 0,Y 559.87,Z 306.295,A -85,B 0,C 180,E1 -2949.999,E2 -2949.999} C_VEL
LIN {X 0,Y 559.62,Z 326.692,A -85,B 0,C 180,E1 -2952.927,E2 -2952.927} C_VEL
LIN {X 0,Y 559.397,Z 346.622,A -85,B 0,C 180,E1 -2955.797,E2 -2955.797} C_VEL
LIN {X 0,Y 560.284,Z 354.396,A -85,B 0,C 180,E1 -2955.936,E2 -2955.936} C_VEL
LIN {X 0,Y 560.035,Z 455.008,A -85,B 0,C 180,E1 -2957.246,E2 -2957.246} C_VEL
LIN {X 0,Y 559.913,Z 468.259,A -85,B 0,C 180,E1 -2957.566,E2 -2957.566} C_VEL
LIN {X 0,Y 559.76,Z 480.408,A -85,B 0,C 180,E1 -2957.999,E2 -2957.999} C_VEL
LIN {X 0,Y 559.667,Z 491.833,A -85,B 0,C 180,E1 -2958.548,E2 -2958.548} C_VEL
LIN {X 0,Y 559.504,Z 502.922,A -85,B 0,C 180,E1 -2959.232,E2 -2959.232} C_VEL
LIN {X 0,Y 559.308,Z 513.552,A -85,B 0,C 180,E1 -2960.052,E2 -2960.052} C_VEL
LIN {X 0,Y 559.16,Z 523.108,A -85,B 0,C 180,E1 -2960.962,E2 -2960.962} C_VEL
LIN {X 0,Y 559.046,Z 530.97,A -85,B 0,C 180,E1 -2961.871,E2 -2961.871} C_VEL
LIN {X 0,Y 558.943,Z 538.63,A -85,B 0,C 180,E1 -2962.96,E2 -2962.96} C_VEL
LIN {X 0,Y 558.935,Z 545.685,A -85,B 0,C 180,E1 -2964.228,E2 -2964.228} C_VEL
LIN {X 0,Y 558.826,Z 550.377,A -85,B 0,C 180,E1 -2965.312,E2 -2965.312} C_VEL
LIN {X 0,Y 558.836,Z 553.961,A -85,B 0,C 180,E1 -2966.396,E2 -2966.396} C_VEL
LIN {X 0,Y 558.799,Z 555.81,A -85,B 0,C 180,E1 -2967.117,E2 -2967.117} C_VEL
LIN {X 0,Y 558.745,Z 558.185,A -85,B 0,C 180,E1 -2968.56,E2 -2968.56} C_VEL
LIN {X 0,Y 558.74,Z 559,A -85,B 0,C 180,E1 -2970.001,E2 -2970.001} C_VEL
LIN {X 0,Y 558.745,Z 558.184,A -85,B 0,C 180,E1 -2971.443,E2 -2971.443} C_VEL
LIN {X 0,Y 558.799,Z 555.808,A -85,B 0,C 180,E1 -2972.885,E2 -2972.885} C_VEL
LIN {X 0,Y 558.844,Z 552.892,A -85,B 0,C 180,E1 -2973.967,E2 -2973.967} C_VEL
LIN {X 0,Y 558.798,Z 548.944,A -85,B 0,C 180,E1 -2975.052,E2 -2975.052} C_VEL
LIN {X 0,Y 558.926,Z 543.862,A -85,B 0,C 180,E1 -2976.136,E2 -2976.136} C_VEL
LIN {X 0,Y 558.978,Z 537.461,A -85,B 0,C 180,E1 -2977.224,E2 -2977.224} C_VEL
LIN {X 0,Y 559.092,Z 529.469,A -85,B 0,C 180,E1 -2978.313,E2 -2978.313} C_VEL
LIN {X 0,Y 559.185,Z 521.325,A -85,B 0,C 180,E1 -2979.222,E2 -2979.222} C_VEL
LIN {X 0,Y 559.337,Z 511.387,A -85,B 0,C 180,E1 -2980.132,E2 -2980.132} C_VEL
LIN {X 0,Y 559.57,Z 500.37,A -85,B 0,C 180,E1 -2980.938,E2 -2980.938} C_VEL
LIN {X 0,Y 559.674,Z 488.441,A -85,B 0,C 180,E1 -2981.629,E2 -2981.629} C_VEL
LIN {X 0,Y 559.797,Z 476.956,A -85,B 0,C 180,E1 -2982.14,E2 -2982.14} C_VEL
LIN {X 0,Y 559.949,Z 464.137,A -85,B 0,C 180,E1 -2982.551,E2 -2982.551} C_VEL
LIN {X 0,Y 560.086,Z 450.539,A -85,B 0,C 180,E1 -2982.824,E2 -2982.824} C_VEL
LIN {X 0,Y 560.199,Z 352.212,A -85,B 0,C 180,E1 -2984.095,E2 -2984.095} C_VEL
LIN {X 0,Y 559.392,Z 346.606,A -85,B 0,C 180,E1 -2984.205,E2 -2984.205} C_VEL
LIN {X 0,Y 559.626,Z 326.677,A -85,B 0,C 180,E1 -2987.075,E2 -2987.075} C_VEL
LIN {X 0,Y 559.891,Z 306.336,A -85,B 0,C 180,E1 -2990.003,E2 -2990.003} C_VEL
LIN {X 0,Y 560.146,Z 287.914,A -85,B 0,C 180,E1 -2992.695,E2 -2992.695} C_VEL
LIN {X 0,Y 559.491,Z 282.603,A -85,B 0,C 180,E1 -2993.51,E2 -2993.51} C_VEL
LIN {X 0,Y 559.162,Z 280.838,A -85,B 0,C 180,E1 -2993.815,E2 -2993.815} C_VEL
LIN {X 0,Y 559.18,Z 280.835,A -85,B 0,C 180,E1 -2996.098,E2 -2996.098} C_VEL
LIN {X 0,Y 559.144,Z 280.833,A -85,B 0,C 180,E1 -2998.532,E2 -2998.532} C_VEL
LIN {X 0,Y 559.151,Z 280.828,A -85,B 0,C 180,E1 -3001.273,E2 -3001.273} C_VEL
LIN {X 0,Y 559.162,Z 280.832,A -85,B 0,C 180,E1 -3003.948,E2 -3003.948} C_VEL
LIN {X 0,Y 559.145,Z 280.829,A -85,B 0,C 180,E1 -3007.109,E2 -3007.109} C_VEL
LIN {X 0,Y 559.164,Z 280.829,A -85,B 0,C 180,E1 -3009.942,E2 -3009.942} C_VEL
LIN {X 0,Y 559.162,Z 280.834,A -85,B 0,C 180,E1 -3012.744,E2 -3012.744} C_VEL
LIN {X 0,Y 559.153,Z 280.828,A -85,B 0,C 180,E1 -3015.762,E2 -3015.762} C_VEL
LIN {X 0,Y 559.168,Z 280.829,A -85,B 0,C 180,E1 -3018.23,E2 -3018.23} C_VEL
LIN {X 0,Y 559.178,Z 280.829,A -85,B 0,C 180,E1 -3021.192,E2 -3021.192} C_VEL
LIN {X 0,Y 559.144,Z 280.829,A -85,B 0,C 180,E1 -3023.789,E2 -3023.789} C_VEL
LIN {X 0,Y 559.151,Z 280.83,A -85,B 0,C 180,E1 -3026.424,E2 -3026.424} C_VEL
LIN {X 0,Y 559.16,Z 280.836,A -85,B 0,C 180,E1 -3028.981,E2 -3028.981} C_VEL
LIN {X 0,Y 559.174,Z 280.829,A -85,B 0,C 180,E1 -3031.619,E2 -3031.619} C_VEL
LIN {X 0,Y 559.182,Z 280.825,A -85,B 0,C 180,E1 -3033.903,E2 -3033.903} C_VEL
LIN {X 0,Y 559.142,Z 280.83,A -85,B 0,C 180,E1 -3036.572,E2 -3036.572} C_VEL
LIN {X 0,Y 559.181,Z 280.835,A -85,B 0,C 180,E1 -3039.395,E2 -3039.395} C_VEL
LIN {X 0,Y 559.141,Z 280.837,A -85,B 0,C 180,E1 -3041.685,E2 -3041.685} C_VEL
LIN {X 0,Y 559.165,Z 280.831,A -85,B 0,C 180,E1 -3043.948,E2 -3043.948} C_VEL
LIN {X 0,Y 559.173,Z 280.828,A -85,B 0,C 180,E1 -3046.184,E2 -3046.184} C_VEL
LIN {X 0,Y 559.197,Z 280.824,A -85,B 0,C 180,E1 -3049.133,E2 -3049.133} C_VEL
LIN {X 0,Y 559.199,Z 280.829,A -85,B 0,C 180,E1 -3052.053,E2 -3052.053} C_VEL
LIN {X 0,Y 559.251,Z 280.816,A -85,B 0,C 180,E1 -3054.953,E2 -3054.953} C_VEL
LIN {X 0,Y 559.257,Z 280.822,A -85,B 0,C 180,E1 -3057.839,E2 -3057.839} C_VEL
LIN {X 0,Y 559.273,Z 280.815,A -85,B 0,C 180,E1 -3060.72,E2 -3060.72} C_VEL
LIN {X 0,Y 559.239,Z 280.818,A -85,B 0,C 180,E1 -3062.881,E2 -3062.881} C_VEL
LIN {X 0,Y 559.226,Z 280.821,A -85,B 0,C 180,E1 -3065.77,E2 -3065.77} C_VEL
LIN {X 0,Y 559.174,Z 280.831,A -85,B 0,C 180,E1 -3068.674,E2 -3068.674} C_VEL
LIN {X 0,Y 559.21,Z 280.821,A -85,B 0,C 180,E1 -3071.6,E2 -3071.6} C_VEL
LIN {X 0,Y 559.205,Z 280.832,A -85,B 0,C 180,E1 -3074.595,E2 -3074.595} C_VEL
LIN {X 0,Y 559.145,Z 280.829,A -85,B 0,C 180,E1 -3077.557,E2 -3077.557} C_VEL
LIN {X 0,Y 559.169,Z 280.826,A -85,B 0,C 180,E1 -3079.837,E2 -3079.837} C_VEL
LIN {X 0,Y 559.143,Z 280.83,A -85,B 0,C 180,E1 -3082.153,E2 -3082.153} C_VEL
LIN {X 0,Y 559.18,Z 280.829,A -85,B 0,C 180,E1 -3085.298,E2 -3085.298} C_VEL
LIN {X 0,Y 559.161,Z 280.828,A -85,B 0,C 180,E1 -3087.713,E2 -3087.713} C_VEL
LIN {X 0,Y 559.143,Z 280.832,A -85,B 0,C 180,E1 -3090.611,E2 -3090.611} C_VEL
LIN {X 0,Y 558.481,Z 280.921,A -85,B 0,C 180,E1 -3091.213,E2 -3091.213} C_VEL
LIN {X 0,Y 555.619,Z 281.279,A -85,B 0,C 180,E1 -3092.189,E2 -3092.189} C_VEL
LIN {X 0,Y 553.206,Z 281.577,A -85,B 0,C 180,E1 -3092.974,E2 -3092.974} C_VEL
LIN {X 0,Y 552.187,Z 281.7,A -85,B 0,C 180,E1 -3093.581,E2 -3093.581} C_VEL
LIN {X 0,Y 552.112,Z 281.707,A -85,B 0,C 180,E1 -3093.786,E2 -3093.786} C_VEL
LIN {X 0,Y 552.102,Z 281.708,A -85,B 0,C 180,E1 -3096.747,E2 -3096.747} C_VEL
LIN {X 0,Y 552.132,Z 281.711,A -85,B 0,C 180,E1 -3099.527,E2 -3099.527} C_VEL
LIN {X 0,Y 552.133,Z 281.702,A -85,B 0,C 180,E1 -3102.425,E2 -3102.425} C_VEL
LIN {X 0,Y 552.095,Z 281.717,A -85,B 0,C 180,E1 -3105.562,E2 -3105.562} C_VEL
LIN {X 0,Y 552.124,Z 281.704,A -85,B 0,C 180,E1 -3108.554,E2 -3108.554} C_VEL
LIN {X 0,Y 552.119,Z 281.708,A -85,B 0,C 180,E1 -3111.41,E2 -3111.41} C_VEL
LIN {X 0,Y 552.088,Z 281.714,A -85,B 0,C 180,E1 -3114.156,E2 -3114.156} C_VEL
LIN {X 0,Y 552.118,Z 281.704,A -85,B 0,C 180,E1 -3116.814,E2 -3116.814} C_VEL
LIN {X 0,Y 552.105,Z 281.707,A -85,B 0,C 180,E1 -3119.39,E2 -3119.39} C_VEL
LIN {X 0,Y 552.124,Z 281.71,A -85,B 0,C 180,E1 -3121.902,E2 -3121.902} C_VEL
LIN {X 0,Y 552.159,Z 281.703,A -85,B 0,C 180,E1 -3124.649,E2 -3124.649} C_VEL
LIN {X 0,Y 552.095,Z 281.708,A -85,B 0,C 180,E1 -3127.548,E2 -3127.548} C_VEL
LIN {X 0,Y 552.152,Z 281.71,A -85,B 0,C 180,E1 -3130.373,E2 -3130.373} C_VEL
LIN {X 0,Y 552.136,Z 281.705,A -85,B 0,C 180,E1 -3132.976,E2 -3132.976} C_VEL
LIN {X 0,Y 552.135,Z 281.704,A -85,B 0,C 180,E1 -3136.004,E2 -3136.004} C_VEL
LIN {X 0,Y 552.163,Z 281.704,A -85,B 0,C 180,E1 -3138.992,E2 -3138.992} C_VEL
LIN {X 0,Y 552.152,Z 281.702,A -85,B 0,C 180,E1 -3141.95,E2 -3141.95} C_VEL
LIN {X 0,Y 552.226,Z 281.702,A -85,B 0,C 180,E1 -3144.888,E2 -3144.888} C_VEL
LIN {X 0,Y 552.141,Z 281.811,A -85,B 0,C 180,E1 -3145.756,E2 -3145.756} C_VEL
LIN {X 0,Y 552.467,Z 286.006,A -85,B 0,C 180,E1 -3146.535,E2 -3146.535} C_VEL
LIN {X 0,Y 552.272,Z 300.876,A -85,B 0,C 180,E1 -3149.27,E2 -3149.27} C_VEL
LIN {X 0,Y 552.106,Z 308.438,A -85,B 0,C 180,E1 -3150.683,E2 -3150.683} C_VEL
LIN {X 0,Y 553.397,Z 315.646,A -85,B 0,C 180,E1 -3150.818,E2 -3150.818} C_VEL
LIN {X 0,Y 553.03,Z 415.574,A -85,B 0,C 180,E1 -3152.138,E2 -3152.138} C_VEL
LIN {X 0,Y 552.904,Z 429.23,A -85,B 0,C 180,E1 -3152.48,E2 -3152.48} C_VEL
LIN {X 0,Y 552.796,Z 442.01,A -85,B 0,C 180,E1 -3152.959,E2 -3152.959} C_VEL
LIN {X 0,Y 552.603,Z 453.704,A -85,B 0,C 180,E1 -3153.553,E2 -3153.553} C_VEL
LIN {X 0,Y 552.38,Z 464.99,A -85,B 0,C 180,E1 -3154.286,E2 -3154.286} C_VEL
LIN {X 0,Y 552.286,Z 475.164,A -85,B 0,C 180,E1 -3155.109,E2 -3155.109} C_VEL
LIN {X 0,Y 552.062,Z 484.383,A -85,B 0,C 180,E1 -3156.028,E2 -3156.028} C_VEL
LIN {X 0,Y 551.966,Z 493.201,A -85,B 0,C 180,E1 -3157.112,E2 -3157.112} C_VEL
LIN {X 0,Y 551.874,Z 500.584,A -85,B 0,C 180,E1 -3158.236,E2 -3158.236} C_VEL
LIN {X 0,Y 551.788,Z 505.496,A -85,B 0,C 180,E1 -3159.16,E2 -3159.16} C_VEL
LIN {X 0,Y 551.747,Z 510.276,A -85,B 0,C 180,E1 -3160.271,E2 -3160.271} C_VEL
LIN {X 0,Y 551.748,Z 513.529,A -85,B 0,C 180,E1 -3161.245,E2 -3161.245} C_VEL
LIN {X 0,Y 551.659,Z 516.576,A -85,B 0,C 180,E1 -3162.507,E2 -3162.507} C_VEL
LIN {X 0,Y 551.655,Z 517.809,A -85,B 0,C 180,E1 -3163.256,E2 -3163.256} C_VEL
LIN {X 0,Y 551.691,Z 518.886,A -85,B 0,C 180,E1 -3164.496,E2 -3164.496} C_VEL
LIN {X 0,Y 551.604,Z 518.903,A -85,B 0,C 180,E1 -3165.518,E2 -3165.518} C_VEL
LIN {X 0,Y 551.63,Z 518.431,A -85,B 0,C 180,E1 -3166.276,E2 -3166.276} C_VEL
LIN {X 0,Y 551.677,Z 517.299,A -85,B 0,C 180,E1 -3167.167,E2 -3167.167} C_VEL
LIN {X 0,Y 551.688,Z 514.326,A -85,B 0,C 180,E1 -3168.569,E2 -3168.569} C_VEL
LIN {X 0,Y 551.771,Z 510.469,A -85,B 0,C 180,E1 -3169.769,E2 -3169.769} C_VEL
LIN {X 0,Y 551.798,Z 505.688,A -85,B 0,C 180,E1 -3170.892,E2 -3170.892} C_VEL
LIN {X 0,Y 551.873,Z 499.306,A -85,B 0,C 180,E1 -3172.065,E2 -3172.065} C_VEL
LIN {X 0,Y 551.976,Z 491.226,A -85,B 0,C 180,E1 -3173.246,E2 -3173.246} C_VEL
LIN {X 0,Y 552.107,Z 482.771,A -85,B 0,C 180,E1 -3174.236,E2 -3174.236} C_VEL
LIN {X 0,Y 552.3,Z 473.115,A -85,B 0,C 180,E1 -3175.158,E2 -3175.158} C_VEL
LIN {X 0,Y 552.458,Z 461.801,A -85,B 0,C 180,E1 -3176.031,E2 -3176.031} C_VEL
LIN {X 0,Y 552.684,Z 450.253,A -85,B 0,C 180,E1 -3176.727,E2 -3176.727} C_VEL
LIN {X 0,Y 552.841,Z 438.293,A -85,B 0,C 180,E1 -3177.285,E2 -3177.285} C_VEL
LIN {X 0,Y 553.012,Z 425.802,A -85,B 0,C 180,E1 -3177.712,E2 -3177.712} C_VEL
LIN {X 0,Y 553.086,Z 413.318,A -85,B 0,C 180,E1 -3177.991,E2 -3177.991} C_VEL
LIN {X 0,Y 553.293,Z 315.196,A -85,B 0,C 180,E1 -3179.281,E2 -3179.281} C_VEL
LIN {X 0,Y 552.192,Z 308.373,A -85,B 0,C 180,E1 -3179.418,E2 -3179.418} C_VEL
LIN {X 0,Y 552.308,Z 292.64,A -85,B 0,C 180,E1 -3182.304,E2 -3182.304} C_VEL
LIN {X 0,Y 552.229,Z 282.726,A -85,B 0,C 180,E1 -3184.052,E2 -3184.052} C_VEL
LIN {X 0,Y 552.067,Z 281.717,A -85,B 0,C 180,E1 -3184.265,E2 -3184.265} C_VEL
LIN {X 0,Y 552.042,Z 281.72,A -85,B 0,C 180,E1 -3186.75,E2 -3186.75} C_VEL
LIN {X 0,Y 552.081,Z 281.717,A -85,B 0,C 180,E1 -3189.529,E2 -3189.529} C_VEL
LIN {X 0,Y 552.067,Z 281.712,A -85,B 0,C 180,E1 -3192.429,E2 -3192.429} C_VEL
LIN {X 0,Y 552.059,Z 281.719,A -85,B 0,C 180,E1 -3195.559,E2 -3195.559} C_VEL
LIN {X 0,Y 552.096,Z 281.717,A -85,B 0,C 180,E1 -3197.586,E2 -3197.586} C_VEL
LIN {X 0,Y 552.111,Z 281.706,A -85,B 0,C 180,E1 -3200.471,E2 -3200.471} C_VEL
LIN {X 0,Y 552.081,Z 281.716,A -85,B 0,C 180,E1 -3203.318,E2 -3203.318} C_VEL
LIN {X 0,Y 552.102,Z 281.713,A -85,B 0,C 180,E1 -3205.937,E2 -3205.937} C_VEL
LIN {X 0,Y 552.106,Z 281.706,A -85,B 0,C 180,E1 -3208.54,E2 -3208.54} C_VEL
LIN {X 0,Y 552.082,Z 281.714,A -85,B 0,C 180,E1 -3211.443,E2 -3211.443} C_VEL
LIN {X 0,Y 552.121,Z 281.704,A -85,B 0,C 180,E1 -3214.654,E2 -3214.654} C_VEL
LIN {X 0,Y 552.075,Z 281.714,A -85,B 0,C 180,E1 -3217.548,E2 -3217.548} C_VEL
LIN {X 0,Y 552.128,Z 281.708,A -85,B 0,C 180,E1 -3220.375,E2 -3220.375} C_VEL
LIN {X 0,Y 552.103,Z 281.705,A -85,B 0,C 180,E1 -3222.976,E2 -3222.976} C_VEL
LIN {X 0,Y 552.114,Z 281.713,A -85,B 0,C 180,E1 -3226.004,E2 -3226.004} C_VEL
LIN {X 0,Y 552.145,Z 281.701,A -85,B 0,C 180,E1 -3228.993,E2 -3228.993} C_VEL
LIN {X 0,Y 552.143,Z 281.706,A -85,B 0,C 180,E1 -3231.951,E2 -3231.951} C_VEL
LIN {X 0,Y 552.209,Z 281.696,A -85,B 0,C 180,E1 -3234.889,E2 -3234.889} C_VEL
LIN {X 0,Y 552.201,Z 281.694,A -85,B 0,C 180,E1 -3237.812,E2 -3237.812} C_VEL
LIN {X 0,Y 552.235,Z 281.696,A -85,B 0,C 180,E1 -3240.729,E2 -3240.729} C_VEL
LIN {X 0,Y 552.199,Z 281.696,A -85,B 0,C 180,E1 -3242.918,E2 -3242.918} C_VEL
LIN {X 0,Y 552.182,Z 281.697,A -85,B 0,C 180,E1 -3245.844,E2 -3245.844} C_VEL
LIN {X 0,Y 552.149,Z 281.708,A -85,B 0,C 180,E1 -3248.786,E2 -3248.786} C_VEL
LIN {X 0,Y 552.151,Z 281.7,A -85,B 0,C 180,E1 -3251.751,E2 -3251.751} C_VEL
LIN {X 0,Y 552.123,Z 281.71,A -85,B 0,C 180,E1 -3254.749,E2 -3254.749} C_VEL
LIN {X 0,Y 552.097,Z 281.706,A -85,B 0,C 180,E1 -3257.789,E2 -3257.789} C_VEL
LIN {X 0,Y 552.117,Z 281.704,A -85,B 0,C 180,E1 -3260.102,E2 -3260.102} C_VEL
LIN {X 0,Y 552.083,Z 281.711,A -85,B 0,C 180,E1 -3262.452,E2 -3262.452} C_VEL
LIN {X 0,Y 552.145,Z 281.708,A -85,B 0,C 180,E1 -3265.352,E2 -3265.352} C_VEL
LIN {X 0,Y 552.112,Z 281.704,A -85,B 0,C 180,E1 -3268.098,E2 -3268.098} C_VEL
LIN {X 0,Y 552.103,Z 281.708,A -85,B 0,C 180,E1 -3270.609,E2 -3270.609} C_VEL
LIN {X 0,Y 552.119,Z 281.712,A -85,B 0,C 180,E1 -3273.186,E2 -3273.186} C_VEL
LIN {X 0,Y 552.103,Z 281.709,A -85,B 0,C 180,E1 -3275.843,E2 -3275.843} C_VEL
LIN {X 0,Y 552.117,Z 281.71,A -85,B 0,C 180,E1 -3279.063,E2 -3279.063} C_VEL
LIN {X 0,Y 552.131,Z 281.714,A -85,B 0,C 180,E1 -3281.445,E2 -3281.445} C_VEL
LIN {X 0,Y 552.088,Z 281.708,A -85,B 0,C 180,E1 -3284.533,E2 -3284.533} C_VEL
LIN {X 0,Y 552.124,Z 281.712,A -85,B 0,C 180,E1 -3287.586,E2 -3287.586} C_VEL
LIN {X 0,Y 552.128,Z 281.704,A -85,B 0,C 180,E1 -3290.475,E2 -3290.475} C_VEL
LIN {X 0,Y 552.114,Z 281.709,A -85,B 0,C 180,E1 -3293.316,E2 -3293.316} C_VEL
LIN {X 0,Y 552.124,Z 281.712,A -85,B 0,C 180,E1 -3295.941,E2 -3295.941} C_VEL
LIN {X 0,Y 552.115,Z 281.707,A -85,B 0,C 180,E1 -3298.542,E2 -3298.542} C_VEL
LIN {X 0,Y 552.122,Z 281.708,A -85,B 0,C 180,E1 -3301.439,E2 -3301.439} C_VEL
LIN {X 0,Y 552.127,Z 281.713,A -85,B 0,C 180,E1 -3304.357,E2 -3304.357} C_VEL
LIN {X 0,Y 552.148,Z 281.802,A -85,B 0,C 180,E1 -3306.117,E2 -3306.117} C_VEL
LIN {X 0,Y 553.191,Z 288.808,A -85,B 0,C 180,E1 -3307.203,E2 -3307.203} C_VEL
LIN {X 0,Y 552.862,Z 310.744,A -85,B 0,C 180,E1 -3310.431,E2 -3310.431} C_VEL
LIN {X 0,Y 552.561,Z 329.709,A -85,B 0,C 180,E1 -3313.182,E2 -3313.182} C_VEL
LIN {X 0,Y 552.372,Z 346.713,A -85,B 0,C 180,E1 -3315.626,E2 -3315.626} C_VEL
LIN {X 0,Y 553.415,Z 354.863,A -85,B 0,C 180,E1 -3315.764,E2 -3315.764} C_VEL
LIN {X 0,Y 553.11,Z 455.008,A -85,B 0,C 180,E1 -3317.084,E2 -3317.084} C_VEL
LIN {X 0,Y 552.993,Z 468.258,A -85,B 0,C 180,E1 -3317.407,E2 -3317.407} C_VEL
LIN {X 0,Y 552.813,Z 481.188,A -85,B 0,C 180,E1 -3317.879,E2 -3317.879} C_VEL
LIN {X 0,Y 552.682,Z 493.647,A -85,B 0,C 180,E1 -3318.507,E2 -3318.507} C_VEL
LIN {X 0,Y 552.466,Z 505.503,A -85,B 0,C 180,E1 -3319.279,E2 -3319.279} C_VEL
LIN {X 0,Y 552.276,Z 515.659,A -85,B 0,C 180,E1 -3320.109,E2 -3320.109} C_VEL
LIN {X 0,Y 552.101,Z 524.796,A -85,B 0,C 180,E1 -3321.03,E2 -3321.03} C_VEL
LIN {X 0,Y 551.959,Z 533.697,A -85,B 0,C 180,E1 -3322.134,E2 -3322.134} C_VEL
LIN {X 0,Y 551.861,Z 539.747,A -85,B 0,C 180,E1 -3323.053,E2 -3323.053} C_VEL
LIN {X 0,Y 551.868,Z 545.685,A -85,B 0,C 180,E1 -3324.154,E2 -3324.154} C_VEL
LIN {X 0,Y 551.725,Z 550.377,A -85,B 0,C 180,E1 -3325.252,E2 -3325.252} C_VEL
LIN {X 0,Y 551.75,Z 553.961,A -85,B 0,C 180,E1 -3326.35,E2 -3326.35} C_VEL
LIN {X 0,Y 551.723,Z 555.81,A -85,B 0,C 180,E1 -3327.08,E2 -3327.08} C_VEL
LIN {X 0,Y 551.644,Z 558.184,A -85,B 0,C 180,E1 -3328.541,E2 -3328.541} C_VEL
LIN {X 0,Y 551.64,Z 559,A -85,B 0,C 180,E1 -3330.001,E2 -3330.001} C_VEL
LIN {X 0,Y 551.645,Z 558.183,A -85,B 0,C 180,E1 -3331.461,E2 -3331.461} C_VEL
LIN {X 0,Y 551.724,Z 555.808,A -85,B 0,C 180,E1 -3332.922,E2 -3332.922} C_VEL
LIN {X 0,Y 551.764,Z 552.892,A -85,B 0,C 180,E1 -3334.018,E2 -3334.018} C_VEL
LIN {X 0,Y 551.724,Z 548.944,A -85,B 0,C 180,E1 -3335.117,E2 -3335.117} C_VEL
LIN {X 0,Y 551.827,Z 543.177,A -85,B 0,C 180,E1 -3336.343,E2 -3336.343} C_VEL
LIN {X 0,Y 551.928,Z 536.229,A -85,B 0,C 180,E1 -3337.501,E2 -3337.501} C_VEL
LIN {X 0,Y 552.065,Z 527.984,A -85,B 0,C 180,E1 -3338.604,E2 -3338.604} C_VEL
LIN {X 0,Y 552.223,Z 519.529,A -85,B 0,C 180,E1 -3339.524,E2 -3339.524} C_VEL
LIN {X 0,Y 552.382,Z 509.08,A -85,B 0,C 180,E1 -3340.447,E2 -3340.447} C_VEL
LIN {X 0,Y 552.614,Z 498.237,A -85,B 0,C 180,E1 -3341.216,E2 -3341.216} C_VEL
LIN {X 0,Y 552.752,Z 487.386,A -85,B 0,C 180,E1 -3341.832,E2 -3341.832} C_VEL
LIN {X 0,Y 552.878,Z 475.737,A -85,B 0,C 180,E1 -3342.341,E2 -3342.341} C_VEL
LIN {X 0,Y 553.007,Z 462.306,A -85,B 0,C 180,E1 -3342.758,E2 -3342.758} C_VEL
LIN {X 0,Y 553.193,Z 449.017,A -85,B 0,C 180,E1 -3343.01,E2 -3343.01} C_VEL
LIN {X 0,Y 553.325,Z 352.907,A -85,B 0,C 180,E1 -3344.264,E2 -3344.264} C_VEL
LIN {X 0,Y 552.388,Z 346.571,A -85,B 0,C 180,E1 -3344.394,E2 -3344.394} C_VEL
LIN {X 0,Y 552.636,Z 325.141,A -85,B 0,C 180,E1 -3347.485,E2 -3347.485} C_VEL
LIN {X 0,Y 552.928,Z 304.77,A -85,B 0,C 180,E1 -3350.46,E2 -3350.46} C_VEL
LIN {X 0,Y 553.143,Z 287.68,A -85,B 0,C 180,E1 -3352.999,E2 -3352.999} C_VEL
LIN {X 0,Y 552.144,Z 281.712,A -85,B 0,C 180,E1 -3353.977,E2 -3353.977} C_VEL
LIN {X 0,Y 552.139,Z 281.704,A -85,B 0,C 180,E1 -3356.999,E2 -3356.999} C_VEL
LIN {X 0,Y 552.121,Z 281.714,A -85,B 0,C 180,E1 -3360.051,E2 -3360.051} C_VEL
LIN {X 0,Y 552.116,Z 281.706,A -85,B 0,C 180,E1 -3362.846,E2 -3362.846} C_VEL
LIN {X 0,Y 552.081,Z 281.709,A -85,B 0,C 180,E1 -3365.44,E2 -3365.44} C_VEL
LIN {X 0,Y 552.1,Z 281.709,A -85,B 0,C 180,E1 -3367.886,E2 -3367.886} C_VEL
LIN {X 0,Y 552.113,Z 281.716,A -85,B 0,C 180,E1 -3370.482,E2 -3370.482} C_VEL
LIN {X 0,Y 552.113,Z 281.705,A -85,B 0,C 180,E1 -3373.424,E2 -3373.424} C_VEL
LIN {X 0,Y 552.113,Z 281.714,A -85,B 0,C 180,E1 -3376.577,E2 -3376.577} C_VEL
LIN {X 0,Y 552.113,Z 281.705,A -85,B 0,C 180,E1 -3379.519,E2 -3379.519} C_VEL
LIN {X 0,Y 552.097,Z 281.709,A -85,B 0,C 180,E1 -3382.336,E2 -3382.336} C_VEL
LIN {X 0,Y 552.087,Z 281.717,A -85,B 0,C 180,E1 -3385.051,E2 -3385.051} C_VEL
LIN {X 0,Y 552.118,Z 281.706,A -85,B 0,C 180,E1 -3387.681,E2 -3387.681} C_VEL
LIN {X 0,Y 552.116,Z 281.704,A -85,B 0,C 180,E1 -3390.235,E2 -3390.235} C_VEL
LIN {X 0,Y 552.142,Z 281.708,A -85,B 0,C 180,E1 -3393,E2 -3393} C_VEL
LIN {X 0,Y 552.118,Z 281.713,A -85,B 0,C 180,E1 -3395.161,E2 -3395.161} C_VEL
LIN {X 0,Y 552.131,Z 281.702,A -85,B 0,C 180,E1 -3398.337,E2 -3398.337} C_VEL
LIN {X 0,Y 552.156,Z 281.7,A -85,B 0,C 180,E1 -3400.674,E2 -3400.674} C_VEL
LIN {X 0,Y 552.116,Z 281.712,A -85,B 0,C 180,E1 -3403.737,E2 -3403.737} C_VEL
LIN {X 0,Y 552.138,Z 281.706,A -85,B 0,C 180,E1 -3406.004,E2 -3406.004} C_VEL
LIN {X 0,Y 552.165,Z 281.699,A -85,B 0,C 180,E1 -3408.993,E2 -3408.993} C_VEL
LIN {X 0,Y 552.154,Z 281.708,A -85,B 0,C 180,E1 -3411.951,E2 -3411.951} C_VEL
LIN {X 0,Y 552.226,Z 281.691,A -85,B 0,C 180,E1 -3414.889,E2 -3414.889} C_VEL
LIN {X 0,Y 552.228,Z 281.697,A -85,B 0,C 180,E1 -3417.812,E2 -3417.812} C_VEL
LIN {X 0,Y 552.244,Z 281.69,A -85,B 0,C 180,E1 -3420.729,E2 -3420.729} C_VEL
LIN {X 0,Y 552.206,Z 281.694,A -85,B 0,C 180,E1 -3422.918,E2 -3422.918} C_VEL
LIN {X 0,Y 552.197,Z 281.698,A -85,B 0,C 180,E1 -3425.844,E2 -3425.844} C_VEL
LIN {X 0,Y 552.145,Z 281.705,A -85,B 0,C 180,E1 -3428.786,E2 -3428.786} C_VEL
LIN {X 0,Y 552.167,Z 281.699,A -85,B 0,C 180,E1 -3431.75,E2 -3431.75} C_VEL
LIN {X 0,Y 552.141,Z 281.709,A -85,B 0,C 180,E1 -3434.748,E2 -3434.748} C_VEL
LIN {X 0,Y 552.102,Z 281.706,A -85,B 0,C 180,E1 -3437.789,E2 -3437.789} C_VEL
LIN {X 0,Y 552.13,Z 281.704,A -85,B 0,C 180,E1 -3440.101,E2 -3440.101} C_VEL
LIN {X 0,Y 552.094,Z 281.711,A -85,B 0,C 180,E1 -3442.451,E2 -3442.451} C_VEL
LIN {X 0,Y 552.16,Z 281.703,A -85,B 0,C 180,E1 -3445.35,E2 -3445.35} C_VEL
LIN {X 0,Y 552.113,Z 281.705,A -85,B 0,C 180,E1 -3448.098,E2 -3448.098} C_VEL
LIN {X 0,Y 552.106,Z 281.708,A -85,B 0,C 180,E1 -3450.609,E2 -3450.609} C_VEL
LIN {X 0,Y 552.119,Z 281.715,A -85,B 0,C 180,E1 -3453.185,E2 -3453.185} C_VEL
LIN {X 0,Y 552.112,Z 281.707,A -85,B 0,C 180,E1 -3453.786,E2 -3453.786} C_VEL
LIN {X 0,Y 551.477,Z 281.786,A -85,B 0,C 180,E1 -3454.395,E2 -3454.395} C_VEL
LIN {X 0,Y 548.652,Z 282.145,A -85,B 0,C 180,E1 -3455.383,E2 -3455.383} C_VEL
LIN {X 0,Y 546.23,Z 282.441,A -85,B 0,C 180,E1 -3456.178,E2 -3456.178} C_VEL
LIN {X 0,Y 545.162,Z 282.574,A -85,B 0,C 180,E1 -3456.792,E2 -3456.792} C_VEL
LIN {X 0,Y 545.06,Z 282.588,A -85,B 0,C 180,E1 -3457,E2 -3457} C_VEL
LIN {X 0,Y 545.068,Z 282.583,A -85,B 0,C 180,E1 -3460.142,E2 -3460.142} C_VEL
LIN {X 0,Y 545.082,Z 282.584,A -85,B 0,C 180,E1 -3463.106,E2 -3463.106} C_VEL
LIN {X 0,Y 545.052,Z 282.586,A -85,B 0,C 180,E1 -3466.226,E2 -3466.226} C_VEL
LIN {X 0,Y 545.085,Z 282.581,A -85,B 0,C 180,E1 -3468.885,E2 -3468.885} C_VEL
LIN {X 0,Y 545.055,Z 282.594,A -85,B 0,C 180,E1 -3471.762,E2 -3471.762} C_VEL
LIN {X 0,Y 545.039,Z 282.587,A -85,B 0,C 180,E1 -3474.531,E2 -3474.531} C_VEL
LIN {X 0,Y 545.072,Z 282.582,A -85,B 0,C 180,E1 -3477.211,E2 -3477.211} C_VEL
LIN {X 0,Y 545.067,Z 282.589,A -85,B 0,C 180,E1 -3479.81,E2 -3479.81} C_VEL
LIN {X 0,Y 545.093,Z 282.587,A -85,B 0,C 180,E1 -3482.344,E2 -3482.344} C_VEL
LIN {X 0,Y 545.121,Z 282.578,A -85,B 0,C 180,E1 -3484.82,E2 -3484.82} C_VEL
LIN {X 0,Y 545.041,Z 282.586,A -85,B 0,C 180,E1 -3487.241,E2 -3487.241} C_VEL
LIN {X 0,Y 545.124,Z 282.586,A -85,B 0,C 180,E1 -3490.414,E2 -3490.414} C_VEL
LIN {X 0,Y 545.068,Z 282.582,A -85,B 0,C 180,E1 -3493.52,E2 -3493.52} C_VEL
LIN {X 0,Y 545.096,Z 282.58,A -85,B 0,C 180,E1 -3495.819,E2 -3495.819} C_VEL
LIN {X 0,Y 545.12,Z 282.584,A -85,B 0,C 180,E1 -3498.848,E2 -3498.848} C_VEL
LIN {X 0,Y 545.1,Z 282.58,A -85,B 0,C 180,E1 -3501.846,E2 -3501.846} C_VEL
LIN {X 0,Y 545.202,Z 282.577,A -85,B 0,C 180,E1 -3504.822,E2 -3504.822} C_VEL
LIN {X 0,Y 545.094,Z 282.695,A -85,B 0,C 180,E1 -3505.678,E2 -3505.678} C_VEL
LIN {X 0,Y 545.46,Z 287.007,A -85,B 0,C 180,E1 -3506.49,E2 -3506.49} C_VEL
LIN {X 0,Y 545.263,Z 302.017,A -85,B 0,C 180,E1 -3509.26,E2 -3509.26} C_VEL
LIN {X 0,Y 545.14,Z 308.524,A -85,B 0,C 180,E1 -3510.484,E2 -3510.484} C_VEL
LIN {X 0,Y 546.552,Z 316.482,A -85,B 0,C 180,E1 -3510.644,E2 -3510.644} C_VEL
LIN {X 0,Y 546.148,Z 415.04,A -85,B 0,C 180,E1 -3511.958,E2 -3511.958} C_VEL
LIN {X 0,Y 546.012,Z 428.192,A -85,B 0,C 180,E1 -3512.281,E2 -3512.281} C_VEL
LIN {X 0,Y 545.876,Z 440.225,A -85,B 0,C 180,E1 -3512.72,E2 -3512.72} C_VEL
LIN {X 0,Y 545.703,Z 452.42,A -85,B 0,C 180,E1 -3513.321,E2 -3513.321} C_VEL
LIN {X 0,Y 545.452,Z 463.934,A -85,B 0,C 180,E1 -3514.063,E2 -3514.063} C_VEL
LIN {X 0,Y 545.267,Z 474.289,A -85,B 0,C 180,E1 -3514.897,E2 -3514.897} C_VEL
LIN {X 0,Y 545.051,Z 482.801,A -85,B 0,C 180,E1 -3515.734,E2 -3515.734} C_VEL
LIN {X 0,Y 544.949,Z 491.432,A -85,B 0,C 180,E1 -3516.765,E2 -3516.765} C_VEL
LIN {X 0,Y 544.829,Z 499.519,A -85,B 0,C 180,E1 -3517.97,E2 -3517.97} C_VEL
LIN {X 0,Y 544.688,Z 506.444,A -85,B 0,C 180,E1 -3519.28,E2 -3519.28} C_VEL
LIN {X 0,Y 544.653,Z 511.012,A -85,B 0,C 180,E1 -3520.406,E2 -3520.406} C_VEL
LIN {X 0,Y 544.652,Z 513.777,A -85,B 0,C 180,E1 -3521.282,E2 -3521.282} C_VEL
LIN {X 0,Y 544.568,Z 516.957,A -85,B 0,C 180,E1 -3522.672,E2 -3522.672} C_VEL
LIN {X 0,Y 544.554,Z 518.038,A -85,B 0,C 180,E1 -3523.432,E2 -3523.432} C_VEL
LIN {X 0,Y 544.588,Z 518.902,A -85,B 0,C 180,E1 -3524.56,E2 -3524.56} C_VEL
LIN {X 0,Y 544.527,Z 518.824,A -85,B 0,C 180,E1 -3525.725,E2 -3525.725} C_VEL
LIN {X 0,Y 544.553,Z 518.215,A -85,B 0,C 180,E1 -3526.494,E2 -3526.494} C_VEL
LIN {X 0,Y 544.573,Z 517.19,A -85,B 0,C 180,E1 -3527.266,E2 -3527.266} C_VEL
LIN {X 0,Y 544.573,Z 515.722,A -85,B 0,C 180,E1 -3528.042,E2 -3528.042} C_VEL
LIN {X 0,Y 544.633,Z 512.598,A -85,B 0,C 180,E1 -3529.21,E2 -3529.21} C_VEL
LIN {X 0,Y 544.683,Z 508.285,A -85,B 0,C 180,E1 -3530.387,E2 -3530.387} C_VEL
LIN {X 0,Y 544.75,Z 501.737,A -85,B 0,C 180,E1 -3531.737,E2 -3531.737} C_VEL
LIN {X 0,Y 544.856,Z 495.431,A -85,B 0,C 180,E1 -3532.764,E2 -3532.764} C_VEL
LIN {X 0,Y 545.019,Z 487.692,A -85,B 0,C 180,E1 -3533.797,E2 -3533.797} C_VEL
LIN {X 0,Y 545.196,Z 477.764,A -85,B 0,C 180,E1 -3534.868,E2 -3534.868} C_VEL
LIN {X 0,Y 545.429,Z 467.888,A -85,B 0,C 180,E1 -3535.729,E2 -3535.729} C_VEL
LIN {X 0,Y 545.586,Z 457.16,A -85,B 0,C 180,E1 -3536.487,E2 -3536.487} C_VEL
LIN {X 0,Y 545.847,Z 446.041,A -85,B 0,C 180,E1 -3537.104,E2 -3537.104} C_VEL
LIN {X 0,Y 546,Z 434.283,A -85,B 0,C 180,E1 -3537.604,E2 -3537.604} C_VEL
LIN {X 0,Y 546.162,Z 420.714,A -85,B 0,C 180,E1 -3538.012,E2 -3538.012} C_VEL
LIN {X 0,Y 546.25,Z 407.799,A -85,B 0,C 180,E1 -3538.242,E2 -3538.242} C_VEL
LIN {X 0,Y 546.459,Z 316.197,A -85,B 0,C 180,E1 -3539.453,E2 -3539.453} C_VEL
LIN {X 0,Y 545.165,Z 308.484,A -85,B 0,C 180,E1 -3539.607,E2 -3539.607} C_VEL
LIN {X 0,Y 545.288,Z 293.543,A -85,B 0,C 180,E1 -3542.334,E2 -3542.334} C_VEL
LIN {X 0,Y 545.255,Z 284.121,A -85,B 0,C 180,E1 -3544.016,E2 -3544.016} C_VEL
LIN {X 0,Y 545.062,Z 282.59,A -85,B 0,C 180,E1 -3544.325,E2 -3544.325} C_VEL
LIN {X 0,Y 545,Z 282.602,A -85,B 0,C 180,E1 -3547.305,E2 -3547.305} C_VEL
LIN {X 0,Y 545.034,Z 282.589,A -85,B 0,C 180,E1 -3550.143,E2 -3550.143} C_VEL
LIN {X 0,Y 544.986,Z 282.601,A -85,B 0,C 180,E1 -3553.114,E2 -3553.114} C_VEL
LIN {X 0,Y 545.032,Z 282.587,A -85,B 0,C 180,E1 -3556.226,E2 -3556.226} C_VEL
LIN {X 0,Y 545.006,Z 282.593,A -85,B 0,C 180,E1 -3558.879,E2 -3558.879} C_VEL
LIN {X 0,Y 545.03,Z 282.596,A -85,B 0,C 180,E1 -3561.761,E2 -3561.761} C_VEL
LIN {X 0,Y 545.009,Z 282.587,A -85,B 0,C 180,E1 -3564.53,E2 -3564.53} C_VEL
LIN {X 0,Y 545.051,Z 282.588,A -85,B 0,C 180,E1 -3567.21,E2 -3567.21} C_VEL
LIN {X 0,Y 545.047,Z 282.596,A -85,B 0,C 180,E1 -3569.81,E2 -3569.81} C_VEL
LIN {X 0,Y 545.03,Z 282.59,A -85,B 0,C 180,E1 -3572.341,E2 -3572.341} C_VEL
LIN {X 0,Y 545.089,Z 282.579,A -85,B 0,C 180,E1 -3574.819,E2 -3574.819} C_VEL
LIN {X 0,Y 545.02,Z 282.59,A -85,B 0,C 180,E1 -3577.242,E2 -3577.242} C_VEL
LIN {X 0,Y 545.1,Z 282.583,A -85,B 0,C 180,E1 -3580.414,E2 -3580.414} C_VEL
LIN {X 0,Y 545.031,Z 282.588,A -85,B 0,C 180,E1 -3583.52,E2 -3583.52} C_VEL
LIN {X 0,Y 545.068,Z 282.588,A -85,B 0,C 180,E1 -3585.819,E2 -3585.819} C_VEL
LIN {X 0,Y 545.101,Z 282.58,A -85,B 0,C 180,E1 -3588.849,E2 -3588.849} C_VEL
LIN {X 0,Y 545.113,Z 282.58,A -85,B 0,C 180,E1 -3591.847,E2 -3591.847} C_VEL
LIN {X 0,Y 545.185,Z 282.572,A -85,B 0,C 180,E1 -3594.823,E2 -3594.823} C_VEL
LIN {X 0,Y 545.173,Z 282.569,A -85,B 0,C 180,E1 -3597.784,E2 -3597.784} C_VEL
LIN {X 0,Y 545.204,Z 282.572,A -85,B 0,C 180,E1 -3600.739,E2 -3600.739} C_VEL
LIN {X 0,Y 545.164,Z 282.572,A -85,B 0,C 180,E1 -3602.956,E2 -3602.956} C_VEL
LIN {X 0,Y 545.153,Z 282.573,A -85,B 0,C 180,E1 -3605.92,E2 -3605.92} C_VEL
LIN {X 0,Y 545.108,Z 282.584,A -85,B 0,C 180,E1 -3608.9,E2 -3608.9} C_VEL
LIN {X 0,Y 545.122,Z 282.576,A -85,B 0,C 180,E1 -3611.905,E2 -3611.905} C_VEL
LIN {X 0,Y 545.072,Z 282.591,A -85,B 0,C 180,E1 -3614.944,E2 -3614.944} C_VEL
LIN {X 0,Y 545.065,Z 282.582,A -85,B 0,C 180,E1 -3618.026,E2 -3618.026} C_VEL
LIN {X 0,Y 545.082,Z 282.582,A -85,B 0,C 180,E1 -3620.373,E2 -3620.373} C_VEL
LIN {X 0,Y 545.079,Z 282.583,A -85,B 0,C 180,E1 -3623.56,E2 -3623.56} C_VEL
LIN {X 0,Y 545.078,Z 282.582,A -85,B 0,C 180,E1 -3626.001,E2 -3626.001} C_VEL
LIN {X 0,Y 545.08,Z 282.583,A -85,B 0,C 180,E1 -3628.75,E2 -3628.75} C_VEL
LIN {X 0,Y 545.067,Z 282.585,A -85,B 0,C 180,E1 -3631.683,E2 -3631.683} C_VEL
LIN {X 0,Y 545.074,Z 282.584,A -85,B 0,C 180,E1 -3634.564,E2 -3634.564} C_VEL
LIN {X 0,Y 545.059,Z 282.593,A -85,B 0,C 180,E1 -3637.302,E2 -3637.302} C_VEL
LIN {X 0,Y 545.067,Z 282.585,A -85,B 0,C 180,E1 -3640.143,E2 -3640.143} C_VEL
LIN {X 0,Y 545.078,Z 282.585,A -85,B 0,C 180,E1 -3643.107,E2 -3643.107} C_VEL
LIN {X 0,Y 545.057,Z 282.584,A -85,B 0,C 180,E1 -3646.226,E2 -3646.226} C_VEL
LIN {X 0,Y 545.095,Z 282.581,A -85,B 0,C 180,E1 -3648.889,E2 -3648.889} C_VEL
LIN {X 0,Y 545.049,Z 282.596,A -85,B 0,C 180,E1 -3651.764,E2 -3651.764} C_VEL
LIN {X 0,Y 545.048,Z 282.588,A -85,B 0,C 180,E1 -3654.534,E2 -3654.534} C_VEL
LIN {X 0,Y 545.064,Z 282.585,A -85,B 0,C 180,E1 -3657.213,E2 -3657.213} C_VEL
LIN {X 0,Y 545.061,Z 282.593,A -85,B 0,C 180,E1 -3659.812,E2 -3659.812} C_VEL
LIN {X 0,Y 545.091,Z 282.587,A -85,B 0,C 180,E1 -3662.346,E2 -3662.346} C_VEL
LIN {X 0,Y 545.115,Z 282.582,A -85,B 0,C 180,E1 -3664.822,E2 -3664.822} C_VEL
LIN {X 0,Y 545.102,Z 282.657,A -85,B 0,C 180,E1 -3665.967,E2 -3665.967} C_VEL
LIN {X 0,Y 546.253,Z 289.823,A -85,B 0,C 180,E1 -3667.097,E2 -3667.097} C_VEL
LIN {X 0,Y 545.887,Z 311.241,A -85,B 0,C 180,E1 -3670.288,E2 -3670.288} C_VEL
LIN {X 0,Y 545.54,Z 330.731,A -85,B 0,C 180,E1 -3673.152,E2 -3673.152} C_VEL
LIN {X 0,Y 545.356,Z 346.417,A -85,B 0,C 180,E1 -3675.435,E2 -3675.435} C_VEL
LIN {X 0,Y 546.543,Z 355.413,A -85,B 0,C 180,E1 -3675.592,E2 -3675.592} C_VEL
LIN {X 0,Y 546.193,Z 454.858,A -85,B 0,C 180,E1 -3676.917,E2 -3676.917} C_VEL
LIN {X 0,Y 546.058,Z 468.14,A -85,B 0,C 180,E1 -3677.245,E2 -3677.245} C_VEL
LIN {X 0,Y 545.858,Z 480.316,A -85,B 0,C 180,E1 -3677.689,E2 -3677.689} C_VEL
LIN {X 0,Y 545.713,Z 492.495,A -85,B 0,C 180,E1 -3678.292,E2 -3678.292} C_VEL
LIN {X 0,Y 545.525,Z 502.918,A -85,B 0,C 180,E1 -3678.953,E2 -3678.953} C_VEL
LIN {X 0,Y 545.278,Z 513.549,A -85,B 0,C 180,E1 -3679.793,E2 -3679.793} C_VEL
LIN {X 0,Y 545.084,Z 523.125,A -85,B 0,C 180,E1 -3680.727,E2 -3680.727} C_VEL
LIN {X 0,Y 544.971,Z 530.97,A -85,B 0,C 180,E1 -3681.659,E2 -3681.659} C_VEL
LIN {X 0,Y 544.823,Z 538.628,A -85,B 0,C 180,E1 -3682.776,E2 -3682.776} C_VEL
LIN {X 0,Y 544.778,Z 545.685,A -85,B 0,C 180,E1 -3684.077,E2 -3684.077} C_VEL
LIN {X 0,Y 544.628,Z 550.377,A -85,B 0,C 180,E1 -3685.19,E2 -3685.19} C_VEL
LIN {X 0,Y 544.668,Z 553.961,A -85,B 0,C 180,E1 -3686.302,E2 -3686.302} C_VEL
LIN {X 0,Y 544.65,Z 555.809,A -85,B 0,C 180,E1 -3687.043,E2 -3687.043} C_VEL
LIN {X 0,Y 544.545,Z 558.183,A -85,B 0,C 180,E1 -3688.522,E2 -3688.522} C_VEL
LIN {X 0,Y 544.541,Z 559,A -85,B 0,C 180,E1 -3690.001,E2 -3690.001} C_VEL
LIN {X 0,Y 544.545,Z 558.182,A -85,B 0,C 180,E1 -3691.48,E2 -3691.48} C_VEL
LIN {X 0,Y 544.651,Z 555.808,A -85,B 0,C 180,E1 -3692.96,E2 -3692.96} C_VEL
LIN {X 0,Y 544.684,Z 552.892,A -85,B 0,C 180,E1 -3694.071,E2 -3694.071} C_VEL
LIN {X 0,Y 544.654,Z 548.944,A -85,B 0,C 180,E1 -3695.183,E2 -3695.183} C_VEL
LIN {X 0,Y 544.74,Z 543.587,A -85,B 0,C 180,E1 -3696.35,E2 -3696.35} C_VEL
LIN {X 0,Y 544.861,Z 536.228,A -85,B 0,C 180,E1 -3697.598,E2 -3697.598} C_VEL
LIN {X 0,Y 545.017,Z 527.984,A -85,B 0,C 180,E1 -3698.716,E2 -3698.716} C_VEL
LIN {X 0,Y 545.203,Z 519.53,A -85,B 0,C 180,E1 -3699.648,E2 -3699.648} C_VEL
LIN {X 0,Y 545.37,Z 509.078,A -85,B 0,C 180,E1 -3700.583,E2 -3700.583} C_VEL
LIN {X 0,Y 545.612,Z 497.475,A -85,B 0,C 180,E1 -3701.411,E2 -3701.411} C_VEL
LIN {X 0,Y 545.797,Z 487.331,A -85,B 0,C 180,E1 -3701.985,E2 -3701.985} C_VEL
LIN {X 0,Y 545.943,Z 475.643,A -85,B 0,C 180,E1 -3702.5,E2 -3702.5} C_VEL
LIN {X 0,Y 546.079,Z 462.177,A -85,B 0,C 180,E1 -3702.922,E2 -3702.922} C_VEL
LIN {X 0,Y 546.264,Z 448.858,A -85,B 0,C 180,E1 -3703.178,E2 -3703.178} C_VEL
LIN {X 0,Y 546.448,Z 353.71,A -85,B 0,C 180,E1 -3704.434,E2 -3704.434} C_VEL
LIN {X 0,Y 545.361,Z 346.44,A -85,B 0,C 180,E1 -3704.567,E2 -3704.567} C_VEL
LIN {X 0,Y 545.652,Z 324.683,A -85,B 0,C 180,E1 -3707.747,E2 -3707.747} C_VEL
LIN {X 0,Y 545.978,Z 304.52,A -85,B 0,C 180,E1 -3710.732,E2 -3710.732} C_VEL
LIN {X 0,Y 546.188,Z 288.76,A -85,B 0,C 180,E1 -3713.108,E2 -3713.108} C_VEL
LIN {X 0,Y 545.116,Z 282.587,A -85,B 0,C 180,E1 -3714.121,E2 -3714.121} C_VEL
LIN {X 0,Y 545.086,Z 282.583,A -85,B 0,C 180,E1 -3717.171,E2 -3717.171} C_VEL
LIN {X 0,Y 545.084,Z 282.591,A -85,B 0,C 180,E1 -3720.247,E2 -3720.247} C_VEL
LIN {X 0,Y 545.079,Z 282.581,A -85,B 0,C 180,E1 -3723.062,E2 -3723.062} C_VEL
LIN {X 0,Y 545.038,Z 282.587,A -85,B 0,C 180,E1 -3725.673,E2 -3725.673} C_VEL
LIN {X 0,Y 545.055,Z 282.592,A -85,B 0,C 180,E1 -3728.238,E2 -3728.238} C_VEL
LIN {X 0,Y 545.086,Z 282.582,A -85,B 0,C 180,E1 -3731.115,E2 -3731.115} C_VEL
LIN {X 0,Y 545.054,Z 282.587,A -85,B 0,C 180,E1 -3734.13,E2 -3734.13} C_VEL
LIN {X 0,Y 545.068,Z 282.584,A -85,B 0,C 180,E1 -3737.304,E2 -3737.304} C_VEL
LIN {X 0,Y 545.07,Z 282.582,A -85,B 0,C 180,E1 -3739.857,E2 -3739.857} C_VEL
LIN {X 0,Y 545.076,Z 282.589,A -85,B 0,C 180,E1 -3743.074,E2 -3743.074} C_VEL
LIN {X 0,Y 545.054,Z 282.585,A -85,B 0,C 180,E1 -3746.327,E2 -3746.327} C_VEL
LIN {X 0,Y 545.071,Z 282.59,A -85,B 0,C 180,E1 -3748.952,E2 -3748.952} C_VEL
LIN {X 0,Y 545.106,Z 282.582,A -85,B 0,C 180,E1 -3751.508,E2 -3751.508} C_VEL
LIN {X 0,Y 545.091,Z 282.58,A -85,B 0,C 180,E1 -3754.493,E2 -3754.493} C_VEL
LIN {X 0,Y 545.041,Z 282.594,A -85,B 0,C 180,E1 -3757.242,E2 -3757.242} C_VEL
LIN {X 0,Y 545.122,Z 282.576,A -85,B 0,C 180,E1 -3760.415,E2 -3760.415} C_VEL
LIN {X 0,Y 545.068,Z 282.593,A -85,B 0,C 180,E1 -3763.521,E2 -3763.521} C_VEL
LIN {X 0,Y 545.099,Z 282.586,A -85,B 0,C 180,E1 -3765.82,E2 -3765.82} C_VEL
LIN {X 0,Y 545.121,Z 282.576,A -85,B 0,C 180,E1 -3768.849,E2 -3768.849} C_VEL
LIN {X 0,Y 545.125,Z 282.586,A -85,B 0,C 180,E1 -3771.847,E2 -3771.847} C_VEL
LIN {X 0,Y 545.202,Z 282.566,A -85,B 0,C 180,E1 -3774.823,E2 -3774.823} C_VEL
LIN {X 0,Y 545.2,Z 282.572,A -85,B 0,C 180,E1 -3777.784,E2 -3777.784} C_VEL
LIN {X 0,Y 545.214,Z 282.566,A -85,B 0,C 180,E1 -3780.738,E2 -3780.738} C_VEL
LIN {X 0,Y 545.173,Z 282.57,A -85,B 0,C 180,E1 -3782.956,E2 -3782.956} C_VEL
LIN {X 0,Y 545.169,Z 282.574,A -85,B 0,C 180,E1 -3785.919,E2 -3785.919} C_VEL
LIN {X 0,Y 545.106,Z 282.58,A -85,B 0,C 180,E1 -3788.9,E2 -3788.9} C_VEL
LIN {X 0,Y 545.111,Z 282.579,A -85,B 0,C 180,E1 -3791.905,E2 -3791.905} C_VEL
LIN {X 0,Y 545.09,Z 282.584,A -85,B 0,C 180,E1 -3794.943,E2 -3794.943} C_VEL
LIN {X 0,Y 545.074,Z 282.583,A -85,B 0,C 180,E1 -3798.026,E2 -3798.026} C_VEL
LIN {X 0,Y 545.096,Z 282.583,A -85,B 0,C 180,E1 -3800.372,E2 -3800.372} C_VEL
LIN {X 0,Y 545.082,Z 282.582,A -85,B 0,C 180,E1 -3803.559,E2 -3803.559} C_VEL
LIN {X 0,Y 545.083,Z 282.581,A -85,B 0,C 180,E1 -3806,E2 -3806} C_VEL
LIN {X 0,Y 545.093,Z 282.585,A -85,B 0,C 180,E1 -3808.748,E2 -3808.748} C_VEL
LIN {X 0,Y 545.062,Z 282.586,A -85,B 0,C 180,E1 -3811.678,E2 -3811.678} C_VEL
LIN {X 0,Y 545.065,Z 282.584,A -85,B 0,C 180,E1 -3814.564,E2 -3814.564} C_VEL
LIN {X 0,Y 545.06,Z 282.588,A -85,B 0,C 180,E1 -3817,E2 -3817} C_VEL
LIN {X 0,Y 544.354,Z 282.682,A -85,B 0,C 180,E1 -3817.616,E2 -3817.616} C_VEL
LIN {X 0,Y 541.491,Z 283.039,A -85,B 0,C 180,E1 -3818.617,E2 -3818.617} C_VEL
LIN {X 0,Y 539.104,Z 283.336,A -85,B 0,C 180,E1 -3819.423,E2 -3819.423} C_VEL
LIN {X 0,Y 538.095,Z 283.453,A -85,B 0,C 180,E1 -3820.045,E2 -3820.045} C_VEL
LIN {X 0,Y 538.02,Z 283.461,A -85,B 0,C 180,E1 -3820.255,E2 -3820.255} C_VEL
LIN {X 0,Y 538.03,Z 283.462,A -85,B 0,C 180,E1 -3822.987,E2 -3822.987} C_VEL
LIN {X 0,Y 538.007,Z 283.464,A -85,B 0,C 180,E1 -3826.183,E2 -3826.183} C_VEL
LIN {X 0,Y 538.052,Z 283.46,A -85,B 0,C 180,E1 -3829.252,E2 -3829.252} C_VEL
LIN {X 0,Y 537.995,Z 283.469,A -85,B 0,C 180,E1 -3832.122,E2 -3832.122} C_VEL
LIN {X 0,Y 538.001,Z 283.463,A -85,B 0,C 180,E1 -3834.915,E2 -3834.915} C_VEL
LIN {X 0,Y 538.022,Z 283.464,A -85,B 0,C 180,E1 -3837.617,E2 -3837.617} C_VEL
LIN {X 0,Y 538.02,Z 283.468,A -85,B 0,C 180,E1 -3840.238,E2 -3840.238} C_VEL
LIN {X 0,Y 538.067,Z 283.456,A -85,B 0,C 180,E1 -3842.795,E2 -3842.795} C_VEL
LIN {X 0,Y 538.031,Z 283.459,A -85,B 0,C 180,E1 -3845.291,E2 -3845.291} C_VEL
LIN {X 0,Y 538.019,Z 283.466,A -85,B 0,C 180,E1 -3848.041,E2 -3848.041} C_VEL
LIN {X 0,Y 538.038,Z 283.461,A -85,B 0,C 180,E1 -3850.939,E2 -3850.939} C_VEL
LIN {X 0,Y 538.02,Z 283.461,A -85,B 0,C 180,E1 -3853.298,E2 -3853.298} C_VEL
LIN {X 0,Y 538.065,Z 283.455,A -85,B 0,C 180,E1 -3855.63,E2 -3855.63} C_VEL
LIN {X 0,Y 538.08,Z 283.464,A -85,B 0,C 180,E1 -3858.701,E2 -3858.701} C_VEL
LIN {X 0,Y 538.064,Z 283.457,A -85,B 0,C 180,E1 -3861.738,E2 -3861.738} C_VEL
LIN {X 0,Y 538.119,Z 283.452,A -85,B 0,C 180,E1 -3864.002,E2 -3864.002} C_VEL
LIN {X 0,Y 538.057,Z 283.606,A -85,B 0,C 180,E1 -3865.598,E2 -3865.598} C_VEL
LIN {X 0,Y 538.451,Z 288.091,A -85,B 0,C 180,E1 -3866.444,E2 -3866.444} C_VEL
LIN {X 0,Y 538.253,Z 303.178,A -85,B 0,C 180,E1 -3869.251,E2 -3869.251} C_VEL
LIN {X 0,Y 538.173,Z 308.841,A -85,B 0,C 180,E1 -3870.303,E2 -3870.303} C_VEL
LIN {X 0,Y 539.679,Z 317.389,A -85,B 0,C 180,E1 -3870.465,E2 -3870.465} C_VEL
LIN {X 0,Y 539.22,Z 415.713,A -85,B 0,C 180,E1 -3871.796,E2 -3871.796} C_VEL
LIN {X 0,Y 539.07,Z 429.47,A -85,B 0,C 180,E1 -3872.147,E2 -3872.147} C_VEL
LIN {X 0,Y 538.958,Z 441.763,A -85,B 0,C 180,E1 -3872.615,E2 -3872.615} C_VEL
LIN {X 0,Y 538.747,Z 452.819,A -85,B 0,C 180,E1 -3873.177,E2 -3873.177} C_VEL
LIN {X 0,Y 538.493,Z 464.299,A -85,B 0,C 180,E1 -3873.928,E2 -3873.928} C_VEL
LIN {X 0,Y 538.271,Z 474.643,A -85,B 0,C 180,E1 -3874.773,E2 -3874.773} C_VEL
LIN {X 0,Y 538.047,Z 483.137,A -85,B 0,C 180,E1 -3875.621,E2 -3875.621} C_VEL
LIN {X 0,Y 537.926,Z 490.88,A -85,B 0,C 180,E1 -3876.552,E2 -3876.552} C_VEL
LIN {X 0,Y 537.786,Z 498.65,A -85,B 0,C 180,E1 -3877.697,E2 -3877.697} C_VEL
LIN {X 0,Y 537.648,Z 505.735,A -85,B 0,C 180,E1 -3879.023,E2 -3879.023} C_VEL
LIN {X 0,Y 537.586,Z 510.462,A -85,B 0,C 180,E1 -3880.164,E2 -3880.164} C_VEL
LIN {X 0,Y 537.57,Z 514.132,A -85,B 0,C 180,E1 -3881.327,E2 -3881.327} C_VEL
LIN {X 0,Y 537.498,Z 515.942,A -85,B 0,C 180,E1 -3882.075,E2 -3882.075} C_VEL
LIN {X 0,Y 537.473,Z 517.327,A -85,B 0,C 180,E1 -3882.842,E2 -3882.842} C_VEL
LIN {X 0,Y 537.472,Z 518.308,A -85,B 0,C 180,E1 -3883.612,E2 -3883.612} C_VEL
LIN {X 0,Y 537.498,Z 518.967,A -85,B 0,C 180,E1 -3884.63,E2 -3884.63} C_VEL
LIN {X 0,Y 537.426,Z 518.747,A -85,B 0,C 180,E1 -3885.938,E2 -3885.938} C_VEL
LIN {X 0,Y 537.471,Z 517.187,A -85,B 0,C 180,E1 -3887.341,E2 -3887.341} C_VEL
LIN {X 0,Y 537.515,Z 514.361,A -85,B 0,C 180,E1 -3888.682,E2 -3888.682} C_VEL
LIN {X 0,Y 537.585,Z 510.678,A -85,B 0,C 180,E1 -3889.87,E2 -3889.87} C_VEL
LIN {X 0,Y 537.649,Z 505.741,A -85,B 0,C 180,E1 -3891.066,E2 -3891.066} C_VEL
LIN {X 0,Y 537.76,Z 499.379,A -85,B 0,C 180,E1 -3892.27,E2 -3892.27} C_VEL
LIN {X 0,Y 537.929,Z 491.321,A -85,B 0,C 180,E1 -3893.482,E2 -3893.482} C_VEL
LIN {X 0,Y 538.092,Z 482.869,A -85,B 0,C 180,E1 -3894.498,E2 -3894.498} C_VEL
LIN {X 0,Y 538.348,Z 472.394,A -85,B 0,C 180,E1 -3895.517,E2 -3895.517} C_VEL
LIN {X 0,Y 538.532,Z 461.887,A -85,B 0,C 180,E1 -3896.339,E2 -3896.339} C_VEL
LIN {X 0,Y 538.809,Z 450.215,A -85,B 0,C 180,E1 -3897.057,E2 -3897.057} C_VEL
LIN {X 0,Y 538.992,Z 438.163,A -85,B 0,C 180,E1 -3897.629,E2 -3897.629} C_VEL
LIN {X 0,Y 539.223,Z 425.57,A -85,B 0,C 180,E1 -3898.061,E2 -3898.061} C_VEL
LIN {X 0,Y 539.284,Z 412.473,A -85,B 0,C 180,E1 -3898.348,E2 -3898.348} C_VEL
LIN {X 0,Y 539.582,Z 316.73,A -85,B 0,C 180,E1 -3899.636,E2 -3899.636} C_VEL
LIN {X 0,Y 538.159,Z 308.57,A -85,B 0,C 180,E1 -3899.805,E2 -3899.805} C_VEL
LIN {X 0,Y 538.264,Z 295.902,A -85,B 0,C 180,E1 -3902.109,E2 -3902.109} C_VEL
LIN {X 0,Y 538.294,Z 285.845,A -85,B 0,C 180,E1 -3903.928,E2 -3903.928} C_VEL
LIN {X 0,Y 538.031,Z 283.467,A -85,B 0,C 180,E1 -3904.389,E2 -3904.389} C_VEL
LIN {X 0,Y 537.962,Z 283.472,A -85,B 0,C 180,E1 -3907.878,E2 -3907.878} C_VEL
LIN {X 0,Y 537.98,Z 283.47,A -85,B 0,C 180,E1 -3910.78,E2 -3910.78} C_VEL
LIN {X 0,Y 537.984,Z 283.468,A -85,B 0,C 180,E1 -3914.07,E2 -3914.07} C_VEL
LIN {X 0,Y 537.967,Z 283.469,A -85,B 0,C 180,E1 -3917.017,E2 -3917.017} C_VEL
LIN {X 0,Y 537.988,Z 283.472,A -85,B 0,C 180,E1 -3919.258,E2 -3919.258} C_VEL
LIN {X 0,Y 537.97,Z 283.471,A -85,B 0,C 180,E1 -3922.121,E2 -3922.121} C_VEL
LIN {X 0,Y 537.99,Z 283.466,A -85,B 0,C 180,E1 -3925.383,E2 -3925.383} C_VEL
LIN {X 0,Y 537.995,Z 283.467,A -85,B 0,C 180,E1 -3928.112,E2 -3928.112} C_VEL
LIN {X 0,Y 538.004,Z 283.464,A -85,B 0,C 180,E1 -3931.097,E2 -3931.097} C_VEL
LIN {X 0,Y 538.001,Z 283.47,A -85,B 0,C 180,E1 -3933.631,E2 -3933.631} C_VEL
LIN {X 0,Y 537.992,Z 283.472,A -85,B 0,C 180,E1 -3936.122,E2 -3936.122} C_VEL
LIN {X 0,Y 538.021,Z 283.46,A -85,B 0,C 180,E1 -3939.348,E2 -3939.348} C_VEL
LIN {X 0,Y 538.02,Z 283.463,A -85,B 0,C 180,E1 -3942.467,E2 -3942.467} C_VEL
LIN {X 0,Y 538.036,Z 283.461,A -85,B 0,C 180,E1 -3945.63,E2 -3945.63} C_VEL
LIN {X 0,Y 538.061,Z 283.458,A -85,B 0,C 180,E1 -3948.701,E2 -3948.701} C_VEL
LIN {X 0,Y 538.07,Z 283.457,A -85,B 0,C 180,E1 -3951.74,E2 -3951.74} C_VEL
LIN {X 0,Y 538.142,Z 283.45,A -85,B 0,C 180,E1 -3954.755,E2 -3954.755} C_VEL
LIN {X 0,Y 538.146,Z 283.445,A -85,B 0,C 180,E1 -3957.755,E2 -3957.755} C_VEL
LIN {X 0,Y 538.173,Z 283.448,A -85,B 0,C 180,E1 -3960.748,E2 -3960.748} C_VEL
LIN {X 0,Y 538.13,Z 283.447,A -85,B 0,C 180,E1 -3962.995,E2 -3962.995} C_VEL
LIN {X 0,Y 538.104,Z 283.452,A -85,B 0,C 180,E1 -3965.998,E2 -3965.998} C_VEL
LIN {X 0,Y 538.059,Z 283.46,A -85,B 0,C 180,E1 -3969.018,E2 -3969.018} C_VEL
LIN {X 0,Y 538.07,Z 283.455,A -85,B 0,C 180,E1 -3972.063,E2 -3972.063} C_VEL
LIN {X 0,Y 538.031,Z 283.465,A -85,B 0,C 180,E1 -3975.144,E2 -3975.144} C_VEL
LIN {X 0,Y 538.018,Z 283.461,A -85,B 0,C 180,E1 -3978.271,E2 -3978.271} C_VEL
LIN {X 0,Y 538.026,Z 283.464,A -85,B 0,C 180,E1 -3980.652,E2 -3980.652} C_VEL
LIN {X 0,Y 538.012,Z 283.461,A -85,B 0,C 180,E1 -3983.888,E2 -3983.888} C_VEL
LIN {X 0,Y 538.039,Z 283.459,A -85,B 0,C 180,E1 -3986.367,E2 -3986.367} C_VEL
LIN {X 0,Y 538.026,Z 283.464,A -85,B 0,C 180,E1 -3988.936,E2 -3988.936} C_VEL
LIN {X 0,Y 538.017,Z 283.461,A -85,B 0,C 180,E1 -3991.891,E2 -3991.891} C_VEL
LIN {X 0,Y 538.024,Z 283.462,A -85,B 0,C 180,E1 -3994.622,E2 -3994.622} C_VEL
LIN {X 0,Y 538.013,Z 283.468,A -85,B 0,C 180,E1 -3997.174,E2 -3997.174} C_VEL
LIN {X 0,Y 538.024,Z 283.466,A -85,B 0,C 180,E1 -3999.797,E2 -3999.797} C_VEL
LIN {X 0,Y 538.015,Z 283.462,A -85,B 0,C 180,E1 -4002.787,E2 -4002.787} C_VEL
LIN {X 0,Y 538.021,Z 283.464,A -85,B 0,C 180,E1 -4005.927,E2 -4005.927} C_VEL
LIN {X 0,Y 538.072,Z 283.459,A -85,B 0,C 180,E1 -4009.25,E2 -4009.25} C_VEL
LIN {X 0,Y 537.989,Z 283.47,A -85,B 0,C 180,E1 -4012.124,E2 -4012.124} C_VEL
LIN {X 0,Y 538.007,Z 283.464,A -85,B 0,C 180,E1 -4014.918,E2 -4014.918} C_VEL
LIN {X 0,Y 538.014,Z 283.468,A -85,B 0,C 180,E1 -4017.619,E2 -4017.619} C_VEL
LIN {X 0,Y 538.014,Z 283.469,A -85,B 0,C 180,E1 -4020.24,E2 -4020.24} C_VEL
LIN {X 0,Y 538.064,Z 283.459,A -85,B 0,C 180,E1 -4022.798,E2 -4022.798} C_VEL
LIN {X 0,Y 538.077,Z 283.548,A -85,B 0,C 180,E1 -4025.82,E2 -4025.82} C_VEL
LIN {X 0,Y 539.289,Z 290.837,A -85,B 0,C 180,E1 -4026.987,E2 -4026.987} C_VEL
LIN {X 0,Y 538.911,Z 312.002,A -85,B 0,C 180,E1 -4030.181,E2 -4030.181} C_VEL
LIN {X 0,Y 538.539,Z 330.444,A -85,B 0,C 180,E1 -4032.926,E2 -4032.926} C_VEL
LIN {X 0,Y 538.319,Z 346.301,A -85,B 0,C 180,E1 -4035.248,E2 -4035.248} C_VEL
LIN {X 0,Y 539.65,Z 355.089,A -85,B 0,C 180,E1 -4035.403,E2 -4035.403} C_VEL
LIN {X 0,Y 539.274,Z 454.542,A -85,B 0,C 180,E1 -4036.746,E2 -4036.746} C_VEL
LIN {X 0,Y 539.152,Z 467.84,A -85,B 0,C 180,E1 -4037.079,E2 -4037.079} C_VEL
LIN {X 0,Y 538.918,Z 480.022,A -85,B 0,C 180,E1 -4037.528,E2 -4037.528} C_VEL
LIN {X 0,Y 538.777,Z 491.561,A -85,B 0,C 180,E1 -4038.101,E2 -4038.101} C_VEL
LIN {X 0,Y 538.532,Z 502.642,A -85,B 0,C 180,E1 -4038.808,E2 -4038.808} C_VEL
LIN {X 0,Y 538.253,Z 513.325,A -85,B 0,C 180,E1 -4039.659,E2 -4039.659} C_VEL
LIN {X 0,Y 538.066,Z 522.957,A -85,B 0,C 180,E1 -4040.605,E2 -4040.605} C_VEL
LIN {X 0,Y 537.911,Z 530.852,A -85,B 0,C 180,E1 -4041.549,E2 -4041.549} C_VEL
LIN {X 0,Y 537.753,Z 538.562,A -85,B 0,C 180,E1 -4042.68,E2 -4042.68} C_VEL
LIN {X 0,Y 537.69,Z 545.672,A -85,B 0,C 180,E1 -4043.999,E2 -4043.999} C_VEL
LIN {X 0,Y 537.54,Z 550.377,A -85,B 0,C 180,E1 -4045.126,E2 -4045.126} C_VEL
LIN {X 0,Y 537.591,Z 553.961,A -85,B 0,C 180,E1 -4046.253,E2 -4046.253} C_VEL
LIN {X 0,Y 537.551,Z 555.809,A -85,B 0,C 180,E1 -4047.003,E2 -4047.003} C_VEL
LIN {X 0,Y 537.451,Z 558.182,A -85,B 0,C 180,E1 -4048.503,E2 -4048.503} C_VEL
LIN {X 0,Y 537.442,Z 559,A -85,B 0,C 180,E1 -4050.001,E2 -4050.001} C_VEL
LIN {X 0,Y 537.451,Z 558.182,A -85,B 0,C 180,E1 -4051.5,E2 -4051.5} C_VEL
LIN {X 0,Y 537.551,Z 555.808,A -85,B 0,C 180,E1 -4052.999,E2 -4052.999} C_VEL
LIN {X 0,Y 537.603,Z 552.892,A -85,B 0,C 180,E1 -4054.124,E2 -4054.124} C_VEL
LIN {X 0,Y 537.588,Z 548.943,A -85,B 0,C 180,E1 -4055.252,E2 -4055.252} C_VEL
LIN {X 0,Y 537.653,Z 544.052,A -85,B 0,C 180,E1 -4056.336,E2 -4056.336} C_VEL
LIN {X 0,Y 537.773,Z 537.386,A -85,B 0,C 180,E1 -4057.51,E2 -4057.51} C_VEL
LIN {X 0,Y 537.943,Z 529.345,A -85,B 0,C 180,E1 -4058.642,E2 -4058.642} C_VEL
LIN {X 0,Y 538.116,Z 521.151,A -85,B 0,C 180,E1 -4059.587,E2 -4059.587} C_VEL
LIN {X 0,Y 538.334,Z 511.159,A -85,B 0,C 180,E1 -4060.532,E2 -4060.532} C_VEL
LIN {X 0,Y 538.594,Z 501.306,A -85,B 0,C 180,E1 -4061.288,E2 -4061.288} C_VEL
LIN {X 0,Y 538.731,Z 490.196,A -85,B 0,C 180,E1 -4061.975,E2 -4061.975} C_VEL
LIN {X 0,Y 538.947,Z 477.71,A -85,B 0,C 180,E1 -4062.57,E2 -4062.57} C_VEL
LIN {X 0,Y 539.139,Z 464.632,A -85,B 0,C 180,E1 -4063.02,E2 -4063.02} C_VEL
LIN {X 0,Y 539.355,Z 451.575,A -85,B 0,C 180,E1 -4063.302,E2 -4063.302} C_VEL
LIN {X 0,Y 539.567,Z 354.283,A -85,B 0,C 180,E1 -4064.611,E2 -4064.611} C_VEL
LIN {X 0,Y 538.34,Z 346.164,A -85,B 0,C 180,E1 -4064.763,E2 -4064.763} C_VEL
LIN {X 0,Y 538.718,Z 323.746,A -85,B 0,C 180,E1 -4068.087,E2 -4068.087} C_VEL
LIN {X 0,Y 539.013,Z 305.595,A -85,B 0,C 180,E1 -4070.813,E2 -4070.813} C_VEL
LIN {X 0,Y 539.314,Z 291.156,A -85,B 0,C 180,E1 -4073.014,E2 -4073.014} C_VEL
LIN {X 0,Y 538.055,Z 283.464,A -85,B 0,C 180,E1 -4074.296,E2 -4074.296} C_VEL
LIN {X 0,Y 538.05,Z 283.46,A -85,B 0,C 180,E1 -4077.35,E2 -4077.35} C_VEL
LIN {X 0,Y 538.033,Z 283.465,A -85,B 0,C 180,E1 -4080.444,E2 -4080.444} C_VEL
LIN {X 0,Y 538.025,Z 283.46,A -85,B 0,C 180,E1 -4083.279,E2 -4083.279} C_VEL
LIN {X 0,Y 538,Z 283.468,A -85,B 0,C 180,E1 -4086.005,E2 -4086.005} C_VEL
LIN {X 0,Y 538.016,Z 283.465,A -85,B 0,C 180,E1 -4088.831,E2 -4088.831} C_VEL
LIN {X 0,Y 538.036,Z 283.459,A -85,B 0,C 180,E1 -4091.774,E2 -4091.774} C_VEL
LIN {X 0,Y 538.01,Z 283.468,A -85,B 0,C 180,E1 -4094.863,E2 -4094.863} C_VEL
LIN {X 0,Y 538.024,Z 283.462,A -85,B 0,C 180,E1 -4097.214,E2 -4097.214} C_VEL
LIN {X 0,Y 538.027,Z 283.461,A -85,B 0,C 180,E1 -4100.203,E2 -4100.203} C_VEL
LIN {X 0,Y 538.03,Z 283.467,A -85,B 0,C 180,E1 -4103.067,E2 -4103.067} C_VEL
LIN {X 0,Y 538.015,Z 283.461,A -85,B 0,C 180,E1 -4105.826,E2 -4105.826} C_VEL
LIN {X 0,Y 538.014,Z 283.463,A -85,B 0,C 180,E1 -4108.499,E2 -4108.499} C_VEL
LIN {X 0,Y 538.049,Z 283.467,A -85,B 0,C 180,E1 -4111.099,E2 -4111.099} C_VEL
LIN {X 0,Y 538.046,Z 283.461,A -85,B 0,C 180,E1 -4113.633,E2 -4113.633} C_VEL
LIN {X 0,Y 538.012,Z 283.462,A -85,B 0,C 180,E1 -4116.122,E2 -4116.122} C_VEL
LIN {X 0,Y 538.042,Z 283.467,A -85,B 0,C 180,E1 -4119.349,E2 -4119.349} C_VEL
LIN {X 0,Y 538.041,Z 283.458,A -85,B 0,C 180,E1 -4122.468,E2 -4122.468} C_VEL
LIN {X 0,Y 538.068,Z 283.465,A -85,B 0,C 180,E1 -4125.631,E2 -4125.631} C_VEL
LIN {X 0,Y 538.081,Z 283.453,A -85,B 0,C 180,E1 -4128.701,E2 -4128.701} C_VEL
LIN {X 0,Y 538.082,Z 283.462,A -85,B 0,C 180,E1 -4131.739,E2 -4131.739} C_VEL
LIN {X 0,Y 538.159,Z 283.443,A -85,B 0,C 180,E1 -4134.755,E2 -4134.755} C_VEL
LIN {X 0,Y 538.172,Z 283.447,A -85,B 0,C 180,E1 -4137.755,E2 -4137.755} C_VEL
LIN {X 0,Y 538.185,Z 283.441,A -85,B 0,C 180,E1 -4140.748,E2 -4140.748} C_VEL
LIN {X 0,Y 538.14,Z 283.446,A -85,B 0,C 180,E1 -4142.994,E2 -4142.994} C_VEL
LIN {X 0,Y 538.12,Z 283.453,A -85,B 0,C 180,E1 -4145.997,E2 -4145.997} C_VEL
LIN {X 0,Y 538.066,Z 283.463,A -85,B 0,C 180,E1 -4148.261,E2 -4148.261} C_VEL
LIN {X 0,Y 538.09,Z 283.452,A -85,B 0,C 180,E1 -4151.598,E2 -4151.598} C_VEL
LIN {X 0,Y 538.064,Z 283.461,A -85,B 0,C 180,E1 -4154.857,E2 -4154.857} C_VEL
LIN {X 0,Y 538.04,Z 283.458,A -85,B 0,C 180,E1 -4157.532,E2 -4157.532} C_VEL
LIN {X 0,Y 538.041,Z 283.466,A -85,B 0,C 180,E1 -4160.651,E2 -4160.651} C_VEL
LIN {X 0,Y 538.005,Z 283.462,A -85,B 0,C 180,E1 -4163.888,E2 -4163.888} C_VEL
LIN {X 0,Y 538.046,Z 283.459,A -85,B 0,C 180,E1 -4166.366,E2 -4166.366} C_VEL
LIN {X 0,Y 538.035,Z 283.467,A -85,B 0,C 180,E1 -4168.933,E2 -4168.933} C_VEL
LIN {X 0,Y 538.014,Z 283.462,A -85,B 0,C 180,E1 -4171.887,E2 -4171.887} C_VEL
LIN {X 0,Y 538.014,Z 283.463,A -85,B 0,C 180,E1 -4174.617,E2 -4174.617} C_VEL
LIN {X 0,Y 538.004,Z 283.47,A -85,B 0,C 180,E1 -4177.169,E2 -4177.169} C_VEL
LIN {X 0,Y 538.02,Z 283.461,A -85,B 0,C 180,E1 -4180.255,E2 -4180.255} C_VEL
LIN {X 0,Y 537.371,Z 283.544,A -85,B 0,C 180,E1 -4180.881,E2 -4180.881} C_VEL
LIN {X 0,Y 534.52,Z 283.908,A -85,B 0,C 180,E1 -4181.896,E2 -4181.896} C_VEL
LIN {X 0,Y 532.094,Z 284.215,A -85,B 0,C 180,E1 -4182.713,E2 -4182.713} C_VEL
LIN {X 0,Y 531.045,Z 284.342,A -85,B 0,C 180,E1 -4183.344,E2 -4183.344} C_VEL
LIN {X 0,Y 530.956,Z 284.349,A -85,B 0,C 180,E1 -4183.558,E2 -4183.558} C_VEL
LIN {X 0,Y 530.957,Z 284.34,A -85,B 0,C 180,E1 -4186.504,E2 -4186.504} C_VEL
LIN {X 0,Y 530.987,Z 284.337,A -85,B 0,C 180,E1 -4188.976,E2 -4188.976} C_VEL
LIN {X 0,Y 530.959,Z 284.346,A -85,B 0,C 180,E1 -4191.529,E2 -4191.529} C_VEL
LIN {X 0,Y 530.957,Z 284.343,A -85,B 0,C 180,E1 -4194.379,E2 -4194.379} C_VEL
LIN {X 0,Y 530.97,Z 284.339,A -85,B 0,C 180,E1 -4197.133,E2 -4197.133} C_VEL
LIN {X 0,Y 530.973,Z 284.344,A -85,B 0,C 180,E1 -4199.802,E2 -4199.802} C_VEL
LIN {X 0,Y 531.019,Z 284.338,A -85,B 0,C 180,E1 -4202.466,E2 -4202.466} C_VEL
LIN {X 0,Y 530.998,Z 284.336,A -85,B 0,C 180,E1 -4204.941,E2 -4204.941} C_VEL
LIN {X 0,Y 530.975,Z 284.347,A -85,B 0,C 180,E1 -4208.246,E2 -4208.246} C_VEL
LIN {X 0,Y 530.997,Z 284.341,A -85,B 0,C 180,E1 -4210.676,E2 -4210.676} C_VEL
LIN {X 0,Y 530.984,Z 284.339,A -85,B 0,C 180,E1 -4213.07,E2 -4213.07} C_VEL
LIN {X 0,Y 531.021,Z 284.333,A -85,B 0,C 180,E1 -4215.435,E2 -4215.435} C_VEL
LIN {X 0,Y 531.039,Z 284.338,A -85,B 0,C 180,E1 -4218.549,E2 -4218.549} C_VEL
LIN {X 0,Y 531.038,Z 284.332,A -85,B 0,C 180,E1 -4221.628,E2 -4221.628} C_VEL
LIN {X 0,Y 531.119,Z 284.33,A -85,B 0,C 180,E1 -4224.684,E2 -4224.684} C_VEL
LIN {X 0,Y 531.003,Z 284.469,A -85,B 0,C 180,E1 -4225.492,E2 -4225.492} C_VEL
LIN {X 0,Y 531.445,Z 289.202,A -85,B 0,C 180,E1 -4226.397,E2 -4226.397} C_VEL
LIN {X 0,Y 531.229,Z 302.375,A -85,B 0,C 180,E1 -4228.862,E2 -4228.862} C_VEL
LIN {X 0,Y 531.183,Z 308.983,A -85,B 0,C 180,E1 -4230.094,E2 -4230.094} C_VEL
LIN {X 0,Y 532.807,Z 318.305,A -85,B 0,C 180,E1 -4230.282,E2 -4230.282} C_VEL
LIN {X 0,Y 532.332,Z 416.333,A -85,B 0,C 180,E1 -4231.63,E2 -4231.63} C_VEL
LIN {X 0,Y 532.16,Z 429.981,A -85,B 0,C 180,E1 -4231.986,E2 -4231.986} C_VEL
LIN {X 0,Y 532.024,Z 442.209,A -85,B 0,C 180,E1 -4232.459,E2 -4232.459} C_VEL
LIN {X 0,Y 531.799,Z 453.213,A -85,B 0,C 180,E1 -4233.029,E2 -4233.029} C_VEL
LIN {X 0,Y 531.506,Z 464.678,A -85,B 0,C 180,E1 -4233.79,E2 -4233.79} C_VEL
LIN {X 0,Y 531.284,Z 474.996,A -85,B 0,C 180,E1 -4234.646,E2 -4234.646} C_VEL
LIN {X 0,Y 531.036,Z 483.477,A -85,B 0,C 180,E1 -4235.505,E2 -4235.505} C_VEL
LIN {X 0,Y 530.878,Z 492.155,A -85,B 0,C 180,E1 -4236.577,E2 -4236.577} C_VEL
LIN {X 0,Y 530.716,Z 500.074,A -85,B 0,C 180,E1 -4237.8,E2 -4237.8} C_VEL
LIN {X 0,Y 530.567,Z 506.925,A -85,B 0,C 180,E1 -4239.145,E2 -4239.145} C_VEL
LIN {X 0,Y 530.508,Z 511.443,A -85,B 0,C 180,E1 -4240.301,E2 -4240.301} C_VEL
LIN {X 0,Y 530.482,Z 514.879,A -85,B 0,C 180,E1 -4241.461,E2 -4241.461} C_VEL
LIN {X 0,Y 530.399,Z 516.591,A -85,B 0,C 180,E1 -4242.239,E2 -4242.239} C_VEL
LIN {X 0,Y 530.373,Z 517.889,A -85,B 0,C 180,E1 -4243.017,E2 -4243.017} C_VEL
LIN {X 0,Y 530.4,Z 518.782,A -85,B 0,C 180,E1 -4243.797,E2 -4243.797} C_VEL
LIN {X 0,Y 530.413,Z 519.247,A -85,B 0,C 180,E1 -4244.703,E2 -4244.703} C_VEL
LIN {X 0,Y 530.332,Z 518.881,A -85,B 0,C 180,E1 -4246.157,E2 -4246.157} C_VEL
LIN {X 0,Y 530.386,Z 517.356,A -85,B 0,C 180,E1 -4247.436,E2 -4247.436} C_VEL
LIN {X 0,Y 530.443,Z 514.044,A -85,B 0,C 180,E1 -4248.94,E2 -4248.94} C_VEL
LIN {X 0,Y 530.522,Z 510.158,A -85,B 0,C 180,E1 -4250.146,E2 -4250.146} C_VEL
LIN {X 0,Y 530.589,Z 505.001,A -85,B 0,C 180,E1 -4251.36,E2 -4251.36} C_VEL
LIN {X 0,Y 530.739,Z 498.393,A -85,B 0,C 180,E1 -4252.581,E2 -4252.581} C_VEL
LIN {X 0,Y 530.923,Z 490.305,A -85,B 0,C 180,E1 -4253.76,E2 -4253.76} C_VEL
LIN {X 0,Y 531.13,Z 481.125,A -85,B 0,C 180,E1 -4254.841,E2 -4254.841} C_VEL
LIN {X 0,Y 531.371,Z 471.356,A -85,B 0,C 180,E1 -4255.772,E2 -4255.772} C_VEL
LIN {X 0,Y 531.599,Z 460.605,A -85,B 0,C 180,E1 -4256.593,E2 -4256.593} C_VEL
LIN {X 0,Y 531.917,Z 448.372,A -85,B 0,C 180,E1 -4257.33,E2 -4257.33} C_VEL
LIN {X 0,Y 532.127,Z 436.413,A -85,B 0,C 180,E1 -4257.876,E2 -4257.876} C_VEL
LIN {X 0,Y 532.309,Z 422.991,A -85,B 0,C 180,E1 -4258.307,E2 -4258.307} C_VEL
LIN {X 0,Y 532.442,Z 410.501,A -85,B 0,C 180,E1 -4258.558,E2 -4258.558} C_VEL
LIN {X 0,Y 532.751,Z 317.837,A -85,B 0,C 180,E1 -4259.816,E2 -4259.816} C_VEL
LIN {X 0,Y 531.177,Z 308.79,A -85,B 0,C 180,E1 -4259.999,E2 -4259.999} C_VEL
LIN {X 0,Y 531.283,Z 294.246,A -85,B 0,C 180,E1 -4262.649,E2 -4262.649} C_VEL
LIN {X 0,Y 531.287,Z 286.851,A -85,B 0,C 180,E1 -4263.977,E2 -4263.977} C_VEL
LIN {X 0,Y 530.98,Z 284.346,A -85,B 0,C 180,E1 -4264.458,E2 -4264.458} C_VEL
LIN {X 0,Y 530.917,Z 284.354,A -85,B 0,C 180,E1 -4267.51,E2 -4267.51} C_VEL
LIN {X 0,Y 530.927,Z 284.347,A -85,B 0,C 180,E1 -4270.436,E2 -4270.436} C_VEL
LIN {X 0,Y 530.907,Z 284.356,A -85,B 0,C 180,E1 -4273.498,E2 -4273.498} C_VEL
LIN {X 0,Y 530.956,Z 284.346,A -85,B 0,C 180,E1 -4275.622,E2 -4275.622} C_VEL
LIN {X 0,Y 530.947,Z 284.343,A -85,B 0,C 180,E1 -4278.56,E2 -4278.56} C_VEL
LIN {X 0,Y 530.936,Z 284.353,A -85,B 0,C 180,E1 -4281.528,E2 -4281.528} C_VEL
LIN {X 0,Y 530.921,Z 284.341,A -85,B 0,C 180,E1 -4284.378,E2 -4284.378} C_VEL
LIN {X 0,Y 530.952,Z 284.344,A -85,B 0,C 180,E1 -4287.133,E2 -4287.133} C_VEL
LIN {X 0,Y 530.954,Z 284.351,A -85,B 0,C 180,E1 -4289.802,E2 -4289.802} C_VEL
LIN {X 0,Y 530.951,Z 284.343,A -85,B 0,C 180,E1 -4292.477,E2 -4292.477} C_VEL
LIN {X 0,Y 530.971,Z 284.338,A -85,B 0,C 180,E1 -4294.941,E2 -4294.941} C_VEL
LIN {X 0,Y 530.956,Z 284.345,A -85,B 0,C 180,E1 -4298.246,E2 -4298.246} C_VEL
LIN {X 0,Y 530.976,Z 284.34,A -85,B 0,C 180,E1 -4300.677,E2 -4300.677} C_VEL
LIN {X 0,Y 530.945,Z 284.34,A -85,B 0,C 180,E1 -4303.07,E2 -4303.07} C_VEL
LIN {X 0,Y 530.993,Z 284.337,A -85,B 0,C 180,E1 -4305.435,E2 -4305.435} C_VEL
LIN {X 0,Y 531.021,Z 284.337,A -85,B 0,C 180,E1 -4308.55,E2 -4308.55} C_VEL
LIN {X 0,Y 531.04,Z 284.332,A -85,B 0,C 180,E1 -4311.629,E2 -4311.629} C_VEL
LIN {X 0,Y 531.101,Z 284.328,A -85,B 0,C 180,E1 -4314.685,E2 -4314.685} C_VEL
LIN {X 0,Y 531.119,Z 284.32,A -85,B 0,C 180,E1 -4317.725,E2 -4317.725} C_VEL
LIN {X 0,Y 531.143,Z 284.323,A -85,B 0,C 180,E1 -4320.758,E2 -4320.758} C_VEL
LIN {X 0,Y 531.095,Z 284.323,A -85,B 0,C 180,E1 -4323.034,E2 -4323.034} C_VEL
LIN {X 0,Y 531.06,Z 284.33,A -85,B 0,C 180,E1 -4326.078,E2 -4326.078} C_VEL
LIN {X 0,Y 531.043,Z 284.333,A -85,B 0,C 180,E1 -4328.371,E2 -4328.371} C_VEL
LIN {X 0,Y 531.044,Z 284.33,A -85,B 0,C 180,E1 -4331.676,E2 -4331.676} C_VEL
LIN {X 0,Y 531.017,Z 284.342,A -85,B 0,C 180,E1 -4334.956,E2 -4334.956} C_VEL
LIN {X 0,Y 531.003,Z 284.334,A -85,B 0,C 180,E1 -4337.723,E2 -4337.723} C_VEL
LIN {X 0,Y 530.987,Z 284.346,A -85,B 0,C 180,E1 -4340.939,E2 -4340.939} C_VEL
LIN {X 0,Y 530.968,Z 284.338,A -85,B 0,C 180,E1 -4344.225,E2 -4344.225} C_VEL
LIN {X 0,Y 531,Z 284.34,A -85,B 0,C 180,E1 -4346.744,E2 -4346.744} C_VEL
LIN {X 0,Y 530.982,Z 284.347,A -85,B 0,C 180,E1 -4349.323,E2 -4349.323} C_VEL
LIN {X 0,Y 530.969,Z 284.338,A -85,B 0,C 180,E1 -4352.104,E2 -4352.104} C_VEL
LIN {X 0,Y 530.98,Z 284.342,A -85,B 0,C 180,E1 -4354.856,E2 -4354.856} C_VEL
LIN {X 0,Y 530.963,Z 284.349,A -85,B 0,C 180,E1 -4357.508,E2 -4357.508} C_VEL
LIN {X 0,Y 530.977,Z 284.34,A -85,B 0,C 180,E1 -4360.434,E2 -4360.434} C_VEL
LIN {X 0,Y 530.959,Z 284.35,A -85,B 0,C 180,E1 -4363.496,E2 -4363.496} C_VEL
LIN {X 0,Y 530.958,Z 284.339,A -85,B 0,C 180,E1 -4366.507,E2 -4366.507} C_VEL
LIN {X 0,Y 531.02,Z 284.341,A -85,B 0,C 180,E1 -4369.573,E2 -4369.573} C_VEL
LIN {X 0,Y 530.964,Z 284.341,A -85,B 0,C 180,E1 -4372.578,E2 -4372.578} C_VEL
LIN {X 0,Y 530.991,Z 284.341,A -85,B 0,C 180,E1 -4375.312,E2 -4375.312} C_VEL
LIN {X 0,Y 530.962,Z 284.347,A -85,B 0,C 180,E1 -4378.033,E2 -4378.033} C_VEL
LIN {X 0,Y 530.986,Z 284.34,A -85,B 0,C 180,E1 -4380.876,E2 -4380.876} C_VEL
LIN {X 0,Y 531.003,Z 284.339,A -85,B 0,C 180,E1 -4383.258,E2 -4383.258} C_VEL
LIN {X 0,Y 531.038,Z 284.501,A -85,B 0,C 180,E1 -4385.676,E2 -4385.676} C_VEL
LIN {X 0,Y 532.329,Z 291.856,A -85,B 0,C 180,E1 -4386.875,E2 -4386.875} C_VEL
LIN {X 0,Y 531.915,Z 313.034,A -85,B 0,C 180,E1 -4390.111,E2 -4390.111} C_VEL
LIN {X 0,Y 531.538,Z 331.48,A -85,B 0,C 180,E1 -4392.892,E2 -4392.892} C_VEL
LIN {X 0,Y 531.301,Z 346.019,A -85,B 0,C 180,E1 -4395.049,E2 -4395.049} C_VEL
LIN {X 0,Y 532.793,Z 357.262,A -85,B 0,C 180,E1 -4395.244,E2 -4395.244} C_VEL
LIN {X 0,Y 532.37,Z 454.226,A -85,B 0,C 180,E1 -4396.571,E2 -4396.571} C_VEL
LIN {X 0,Y 532.228,Z 467.538,A -85,B 0,C 180,E1 -4396.908,E2 -4396.908} C_VEL
LIN {X 0,Y 531.971,Z 479.727,A -85,B 0,C 180,E1 -4397.362,E2 -4397.362} C_VEL
LIN {X 0,Y 531.813,Z 491.212,A -85,B 0,C 180,E1 -4397.939,E2 -4397.939} C_VEL
LIN {X 0,Y 531.556,Z 502.358,A -85,B 0,C 180,E1 -4398.659,E2 -4398.659} C_VEL
LIN {X 0,Y 531.263,Z 513.045,A -85,B 0,C 180,E1 -4399.521,E2 -4399.521} C_VEL
LIN {X 0,Y 531.018,Z 522.677,A -85,B 0,C 180,E1 -4400.479,E2 -4400.479} C_VEL
LIN {X 0,Y 530.849,Z 530.575,A -85,B 0,C 180,E1 -4401.436,E2 -4401.436} C_VEL
LIN {X 0,Y 530.673,Z 538.288,A -85,B 0,C 180,E1 -4402.582,E2 -4402.582} C_VEL
LIN {X 0,Y 530.584,Z 545.4,A -85,B 0,C 180,E1 -4403.918,E2 -4403.918} C_VEL
LIN {X 0,Y 530.459,Z 550.128,A -85,B 0,C 180,E1 -4405.061,E2 -4405.061} C_VEL
LIN {X 0,Y 530.516,Z 553.746,A -85,B 0,C 180,E1 -4406.203,E2 -4406.203} C_VEL
LIN {X 0,Y 530.457,Z 555.609,A -85,B 0,C 180,E1 -4406.963,E2 -4406.963} C_VEL
LIN {X 0,Y 530.41,Z 557.005,A -85,B 0,C 180,E1 -4407.723,E2 -4407.723} C_VEL
LIN {X 0,Y 530.344,Z 558.609,A -85,B 0,C 180,E1 -4409.242,E2 -4409.242} C_VEL
LIN {X 0,Y 530.345,Z 558.826,A -85,B 0,C 180,E1 -4410.001,E2 -4410.001} C_VEL
LIN {X 0,Y 530.361,Z 558.001,A -85,B 0,C 180,E1 -4411.52,E2 -4411.52} C_VEL
LIN {X 0,Y 530.41,Z 557.006,A -85,B 0,C 180,E1 -4412.279,E2 -4412.279} C_VEL
LIN {X 0,Y 530.457,Z 555.61,A -85,B 0,C 180,E1 -4413.039,E2 -4413.039} C_VEL
LIN {X 0,Y 530.523,Z 552.672,A -85,B 0,C 180,E1 -4414.179,E2 -4414.179} C_VEL
LIN {X 0,Y 530.525,Z 548.69,A -85,B 0,C 180,E1 -4415.322,E2 -4415.322} C_VEL
LIN {X 0,Y 530.567,Z 543.127,A -85,B 0,C 180,E1 -4416.551,E2 -4416.551} C_VEL
LIN {X 0,Y 530.731,Z 535.88,A -85,B 0,C 180,E1 -4417.802,E2 -4417.802} C_VEL
LIN {X 0,Y 530.911,Z 527.582,A -85,B 0,C 180,E1 -4418.949,E2 -4418.949} C_VEL
LIN {X 0,Y 531.106,Z 519.076,A -85,B 0,C 180,E1 -4419.907,E2 -4419.907} C_VEL
LIN {X 0,Y 531.359,Z 508.567,A -85,B 0,C 180,E1 -4420.865,E2 -4420.865} C_VEL
LIN {X 0,Y 531.627,Z 497.739,A -85,B 0,C 180,E1 -4421.661,E2 -4421.661} C_VEL
LIN {X 0,Y 531.869,Z 486.777,A -85,B 0,C 180,E1 -4422.303,E2 -4422.303} C_VEL
LIN {X 0,Y 532.045,Z 475.073,A -85,B 0,C 180,E1 -4422.832,E2 -4422.832} C_VEL
LIN {X 0,Y 532.276,Z 461.591,A -85,B 0,C 180,E1 -4423.264,E2 -4423.264} C_VEL
LIN {X 0,Y 532.453,Z 448.217,A -85,B 0,C 180,E1 -4423.526,E2 -4423.526} C_VEL
LIN {X 0,Y 532.76,Z 355.429,A -85,B 0,C 180,E1 -4424.782,E2 -4424.782} C_VEL
LIN {X 0,Y 531.326,Z 345.871,A -85,B 0,C 180,E1 -4424.967,E2 -4424.967} C_VEL
LIN {X 0,Y 531.721,Z 323.659,A -85,B 0,C 180,E1 -4428.307,E2 -4428.307} C_VEL
LIN {X 0,Y 532.129,Z 304.047,A -85,B 0,C 180,E1 -4431.298,E2 -4431.298} C_VEL
LIN {X 0,Y 532.364,Z 292.222,A -85,B 0,C 180,E1 -4433.126,E2 -4433.126} C_VEL
LIN {X 0,Y 531.032,Z 284.338,A -85,B 0,C 180,E1 -4434.431,E2 -4434.431} C_VEL
LIN {X 0,Y 531.015,Z 284.339,A -85,B 0,C 180,E1 -4437.596,E2 -4437.596} C_VEL
LIN {X 0,Y 530.98,Z 284.34,A -85,B 0,C 180,E1 -4440.646,E2 -4440.646} C_VEL
LIN {X 0,Y 530.963,Z 284.342,A -85,B 0,C 180,E1 -4443.775,E2 -4443.775} C_VEL
LIN {X 0,Y 530.96,Z 284.347,A -85,B 0,C 180,E1 -4446.559,E2 -4446.559} C_VEL
LIN {X 0,Y 530.976,Z 284.338,A -85,B 0,C 180,E1 -4449.445,E2 -4449.445} C_VEL
LIN {X 0,Y 530.984,Z 284.346,A -85,B 0,C 180,E1 -4452.457,E2 -4452.457} C_VEL
LIN {X 0,Y 530.981,Z 284.337,A -85,B 0,C 180,E1 -4455.623,E2 -4455.623} C_VEL
LIN {X 0,Y 530.999,Z 284.342,A -85,B 0,C 180,E1 -4458.565,E2 -4458.565} C_VEL
LIN {X 0,Y 530.96,Z 284.341,A -85,B 0,C 180,E1 -4461.529,E2 -4461.529} C_VEL
LIN {X 0,Y 530.959,Z 284.342,A -85,B 0,C 180,E1 -4464.38,E2 -4464.38} C_VEL
LIN {X 0,Y 530.972,Z 284.347,A -85,B 0,C 180,E1 -4467.133,E2 -4467.133} C_VEL
LIN {X 0,Y 530.975,Z 284.339,A -85,B 0,C 180,E1 -4469.803,E2 -4469.803} C_VEL
LIN {X 0,Y 531.017,Z 284.334,A -85,B 0,C 180,E1 -4472.468,E2 -4472.468} C_VEL
LIN {X 0,Y 531.004,Z 284.339,A -85,B 0,C 180,E1 -4474.942,E2 -4474.942} C_VEL
LIN {X 0,Y 530.977,Z 284.338,A -85,B 0,C 180,E1 -4478.247,E2 -4478.247} C_VEL
LIN {X 0,Y 530.996,Z 284.336,A -85,B 0,C 180,E1 -4480.677,E2 -4480.677} C_VEL
LIN {X 0,Y 530.974,Z 284.341,A -85,B 0,C 180,E1 -4483.07,E2 -4483.07} C_VEL
LIN {X 0,Y 531.024,Z 284.339,A -85,B 0,C 180,E1 -4485.436,E2 -4485.436} C_VEL
LIN {X 0,Y 531.039,Z 284.33,A -85,B 0,C 180,E1 -4488.55,E2 -4488.55} C_VEL
LIN {X 0,Y 531.052,Z 284.335,A -85,B 0,C 180,E1 -4491.629,E2 -4491.629} C_VEL
LIN {X 0,Y 531.118,Z 284.321,A -85,B 0,C 180,E1 -4494.685,E2 -4494.685} C_VEL
LIN {X 0,Y 531.144,Z 284.322,A -85,B 0,C 180,E1 -4497.725,E2 -4497.725} C_VEL
LIN {X 0,Y 531.155,Z 284.317,A -85,B 0,C 180,E1 -4500.758,E2 -4500.758} C_VEL
LIN {X 0,Y 531.106,Z 284.322,A -85,B 0,C 180,E1 -4503.034,E2 -4503.034} C_VEL
LIN {X 0,Y 531.077,Z 284.332,A -85,B 0,C 180,E1 -4506.077,E2 -4506.077} C_VEL
LIN {X 0,Y 531.02,Z 284.333,A -85,B 0,C 180,E1 -4509.138,E2 -4509.138} C_VEL
LIN {X 0,Y 531.054,Z 284.329,A -85,B 0,C 180,E1 -4511.67,E2 -4511.67} C_VEL
LIN {X 0,Y 531.036,Z 284.335,A -85,B 0,C 180,E1 -4514.955,E2 -4514.955} C_VEL
LIN {X 0,Y 530.986,Z 284.337,A -85,B 0,C 180,E1 -4517.723,E2 -4517.723} C_VEL
LIN {X 0,Y 531.029,Z 284.333,A -85,B 0,C 180,E1 -4520.127,E2 -4520.127} C_VEL
LIN {X 0,Y 530.949,Z 284.347,A -85,B 0,C 180,E1 -4522.573,E2 -4522.573} C_VEL
LIN {X 0,Y 531.009,Z 284.342,A -85,B 0,C 180,E1 -4525.057,E2 -4525.057} C_VEL
LIN {X 0,Y 531.017,Z 284.335,A -85,B 0,C 180,E1 -4527.595,E2 -4527.595} C_VEL
LIN {X 0,Y 530.978,Z 284.341,A -85,B 0,C 180,E1 -4530.645,E2 -4530.645} C_VEL
LIN {X 0,Y 530.991,Z 284.338,A -85,B 0,C 180,E1 -4533.772,E2 -4533.772} C_VEL
LIN {X 0,Y 530.954,Z 284.341,A -85,B 0,C 180,E1 -4536.558,E2 -4536.558} C_VEL
LIN {X 0,Y 530.988,Z 284.346,A -85,B 0,C 180,E1 -4539.443,E2 -4539.443} C_VEL
LIN {X 0,Y 530.981,Z 284.337,A -85,B 0,C 180,E1 -4542.456,E2 -4542.456} C_VEL
LIN {X 0,Y 530.956,Z 284.349,A -85,B 0,C 180,E1 -4543.558,E2 -4543.558} C_VEL
LIN {X 0,Y 530.282,Z 284.427,A -85,B 0,C 180,E1 -4544.191,E2 -4544.191} C_VEL
LIN {X 0,Y 527.435,Z 284.783,A -85,B 0,C 180,E1 -4545.22,E2 -4545.22} C_VEL
LIN {X 0,Y 525.034,Z 285.082,A -85,B 0,C 180,E1 -4546.048,E2 -4546.048} C_VEL
LIN {X 0,Y 524.003,Z 285.207,A -85,B 0,C 180,E1 -4546.688,E2 -4546.688} C_VEL
LIN {X 0,Y 523.918,Z 285.218,A -85,B 0,C 180,E1 -4546.904,E2 -4546.904} C_VEL
LIN {X 0,Y 523.952,Z 285.22,A -85,B 0,C 180,E1 -4549.92,E2 -4549.92} C_VEL
LIN {X 0,Y 523.91,Z 285.218,A -85,B 0,C 180,E1 -4552.867,E2 -4552.867} C_VEL
LIN {X 0,Y 523.936,Z 285.221,A -85,B 0,C 180,E1 -4555.709,E2 -4555.709} C_VEL
LIN {X 0,Y 523.924,Z 285.22,A -85,B 0,C 180,E1 -4558.455,E2 -4558.455} C_VEL
LIN {X 0,Y 523.943,Z 285.214,A -85,B 0,C 180,E1 -4561.125,E2 -4561.125} C_VEL
LIN {X 0,Y 523.988,Z 285.215,A -85,B 0,C 180,E1 -4563.979,E2 -4563.979} C_VEL
LIN {X 0,Y 523.914,Z 285.218,A -85,B 0,C 180,E1 -4567.106,E2 -4567.106} C_VEL
LIN {X 0,Y 523.982,Z 285.211,A -85,B 0,C 180,E1 -4569.865,E2 -4569.865} C_VEL
LIN {X 0,Y 523.967,Z 285.216,A -85,B 0,C 180,E1 -4572.836,E2 -4572.836} C_VEL
LIN {X 0,Y 523.98,Z 285.211,A -85,B 0,C 180,E1 -4575.235,E2 -4575.235} C_VEL
LIN {X 0,Y 524.015,Z 285.211,A -85,B 0,C 180,E1 -4578.393,E2 -4578.393} C_VEL
LIN {X 0,Y 523.99,Z 285.211,A -85,B 0,C 180,E1 -4581.515,E2 -4581.515} C_VEL
LIN {X 0,Y 524.037,Z 285.206,A -85,B 0,C 180,E1 -4583.84,E2 -4583.84} C_VEL
LIN {X 0,Y 523.994,Z 285.347,A -85,B 0,C 180,E1 -4585.383,E2 -4585.383} C_VEL
LIN {X 0,Y 524.465,Z 290.368,A -85,B 0,C 180,E1 -4586.349,E2 -4586.349} C_VEL
LIN {X 0,Y 524.242,Z 304.639,A -85,B 0,C 180,E1 -4589.039,E2 -4589.039} C_VEL
LIN {X 0,Y 524.22,Z 309.252,A -85,B 0,C 180,E1 -4589.903,E2 -4589.903} C_VEL
LIN {X 0,Y 525.955,Z 319.193,A -85,B 0,C 180,E1 -4590.095,E2 -4590.095} C_VEL
LIN {X 0,Y 525.45,Z 415.842,A -85,B 0,C 180,E1 -4591.436,E2 -4591.436} C_VEL
LIN {X 0,Y 525.295,Z 428.973,A -85,B 0,C 180,E1 -4591.772,E2 -4591.772} C_VEL
LIN {X 0,Y 525.113,Z 441.559,A -85,B 0,C 180,E1 -4592.252,E2 -4592.252} C_VEL
LIN {X 0,Y 524.863,Z 453.603,A -85,B 0,C 180,E1 -4592.877,E2 -4592.877} C_VEL
LIN {X 0,Y 524.53,Z 465.053,A -85,B 0,C 180,E1 -4593.648,E2 -4593.648} C_VEL
LIN {X 0,Y 524.278,Z 475.356,A -85,B 0,C 180,E1 -4594.516,E2 -4594.516} C_VEL
LIN {X 0,Y 524.031,Z 483.816,A -85,B 0,C 180,E1 -4595.386,E2 -4595.386} C_VEL
LIN {X 0,Y 523.848,Z 491.831,A -85,B 0,C 180,E1 -4596.381,E2 -4596.381} C_VEL
LIN {X 0,Y 523.713,Z 499.269,A -85,B 0,C 180,E1 -4597.517,E2 -4597.517} C_VEL
LIN {X 0,Y 523.54,Z 506.338,A -85,B 0,C 180,E1 -4598.879,E2 -4598.879} C_VEL
LIN {X 0,Y 523.437,Z 511.052,A -85,B 0,C 180,E1 -4600.051,E2 -4600.051} C_VEL
LIN {X 0,Y 523.421,Z 515.176,A -85,B 0,C 180,E1 -4601.429,E2 -4601.429} C_VEL
LIN {X 0,Y 523.295,Z 517.24,A -85,B 0,C 180,E1 -4602.407,E2 -4602.407} C_VEL
LIN {X 0,Y 523.28,Z 518.443,A -85,B 0,C 180,E1 -4603.197,E2 -4603.197} C_VEL
LIN {X 0,Y 523.299,Z 519.186,A -85,B 0,C 180,E1 -4603.988,E2 -4603.988} C_VEL
LIN {X 0,Y 523.334,Z 519.527,A -85,B 0,C 180,E1 -4604.781,E2 -4604.781} C_VEL
LIN {X 0,Y 523.247,Z 519.476,A -85,B 0,C 180,E1 -4605.581,E2 -4605.581} C_VEL
LIN {X 0,Y 523.238,Z 518.978,A -85,B 0,C 180,E1 -4606.382,E2 -4606.382} C_VEL
LIN {X 0,Y 523.3,Z 517.517,A -85,B 0,C 180,E1 -4607.534,E2 -4607.534} C_VEL
LIN {X 0,Y 523.395,Z 513.727,A -85,B 0,C 180,E1 -4609.205,E2 -4609.205} C_VEL
LIN {X 0,Y 523.471,Z 509.639,A -85,B 0,C 180,E1 -4610.429,E2 -4610.429} C_VEL
LIN {X 0,Y 523.529,Z 504.235,A -85,B 0,C 180,E1 -4611.663,E2 -4611.663} C_VEL
LIN {X 0,Y 523.717,Z 497.29,A -85,B 0,C 180,E1 -4612.901,E2 -4612.901} C_VEL
LIN {X 0,Y 523.925,Z 489.892,A -85,B 0,C 180,E1 -4613.967,E2 -4613.967} C_VEL
LIN {X 0,Y 524.167,Z 480.322,A -85,B 0,C 180,E1 -4615.087,E2 -4615.087} C_VEL
LIN {X 0,Y 524.487,Z 470.081,A -85,B 0,C 180,E1 -4616.042,E2 -4616.042} C_VEL
LIN {X 0,Y 524.702,Z 459.021,A -85,B 0,C 180,E1 -4616.874,E2 -4616.874} C_VEL
LIN {X 0,Y 525.06,Z 447.465,A -85,B 0,C 180,E1 -4617.555,E2 -4617.555} C_VEL
LIN {X 0,Y 525.257,Z 434.771,A -85,B 0,C 180,E1 -4618.118,E2 -4618.118} C_VEL
LIN {X 0,Y 525.454,Z 421.269,A -85,B 0,C 180,E1 -4618.536,E2 -4618.536} C_VEL
LIN {X 0,Y 525.579,Z 408.164,A -85,B 0,C 180,E1 -4618.774,E2 -4618.774} C_VEL
LIN {X 0,Y 525.832,Z 318.229,A -85,B 0,C 180,E1 -4620.013,E2 -4620.013} C_VEL
LIN {X 0,Y 524.173,Z 308.999,A -85,B 0,C 180,E1 -4620.212,E2 -4620.212} C_VEL
LIN {X 0,Y 524.287,Z 294.313,A -85,B 0,C 180,E1 -4622.879,E2 -4622.879} C_VEL
LIN {X 0,Y 524.151,Z 286.623,A -85,B 0,C 180,E1 -4624.272,E2 -4624.272} C_VEL
LIN {X 0,Y 523.924,Z 285.226,A -85,B 0,C 180,E1 -4624.58,E2 -4624.58} C_VEL
LIN {X 0,Y 523.88,Z 285.226,A -85,B 0,C 180,E1 -4628.103,E2 -4628.103} C_VEL
LIN {X 0,Y 523.875,Z 285.23,A -85,B 0,C 180,E1 -4631.096,E2 -4631.096} C_VEL
LIN {X 0,Y 523.903,Z 285.221,A -85,B 0,C 180,E1 -4634.23,E2 -4634.23} C_VEL
LIN {X 0,Y 523.877,Z 285.223,A -85,B 0,C 180,E1 -4636.829,E2 -4636.829} C_VEL
LIN {X 0,Y 523.899,Z 285.225,A -85,B 0,C 180,E1 -4639.916,E2 -4639.916} C_VEL
LIN {X 0,Y 523.867,Z 285.226,A -85,B 0,C 180,E1 -4642.865,E2 -4642.865} C_VEL
LIN {X 0,Y 523.903,Z 285.226,A -85,B 0,C 180,E1 -4645.708,E2 -4645.708} C_VEL
LIN {X 0,Y 523.906,Z 285.219,A -85,B 0,C 180,E1 -4648.455,E2 -4648.455} C_VEL
LIN {X 0,Y 523.911,Z 285.22,A -85,B 0,C 180,E1 -4651.124,E2 -4651.124} C_VEL
LIN {X 0,Y 523.911,Z 285.226,A -85,B 0,C 180,E1 -4653.993,E2 -4653.993} C_VEL
LIN {X 0,Y 523.897,Z 285.225,A -85,B 0,C 180,E1 -4656.269,E2 -4656.269} C_VEL
LIN {X 0,Y 523.929,Z 285.215,A -85,B 0,C 180,E1 -4658.766,E2 -4658.766} C_VEL
LIN {X 0,Y 523.932,Z 285.217,A -85,B 0,C 180,E1 -4661.22,E2 -4661.22} C_VEL
LIN {X 0,Y 523.902,Z 285.221,A -85,B 0,C 180,E1 -4663.638,E2 -4663.638} C_VEL
LIN {X 0,Y 523.916,Z 285.226,A -85,B 0,C 180,E1 -4666.028,E2 -4666.028} C_VEL
LIN {X 0,Y 523.997,Z 285.214,A -85,B 0,C 180,E1 -4668.394,E2 -4668.394} C_VEL
LIN {X 0,Y 523.988,Z 285.21,A -85,B 0,C 180,E1 -4671.516,E2 -4671.516} C_VEL
LIN {X 0,Y 524.062,Z 285.206,A -85,B 0,C 180,E1 -4674.614,E2 -4674.614} C_VEL
LIN {X 0,Y 524.092,Z 285.195,A -85,B 0,C 180,E1 -4677.695,E2 -4677.695} C_VEL
LIN {X 0,Y 524.112,Z 285.199,A -85,B 0,C 180,E1 -4680.768,E2 -4680.768} C_VEL
LIN {X 0,Y 524.061,Z 285.199,A -85,B 0,C 180,E1 -4683.075,E2 -4683.075} C_VEL
LIN {X 0,Y 524.022,Z 285.207,A -85,B 0,C 180,E1 -4686.159,E2 -4686.159} C_VEL
LIN {X 0,Y 523.991,Z 285.213,A -85,B 0,C 180,E1 -4688.484,E2 -4688.484} C_VEL
LIN {X 0,Y 523.994,Z 285.208,A -85,B 0,C 180,E1 -4691.743,E2 -4691.743} C_VEL
LIN {X 0,Y 523.979,Z 285.217,A -85,B 0,C 180,E1 -4695.053,E2 -4695.053} C_VEL
LIN {X 0,Y 523.95,Z 285.212,A -85,B 0,C 180,E1 -4697.97,E2 -4697.97} C_VEL
LIN {X 0,Y 523.959,Z 285.214,A -85,B 0,C 180,E1 -4700.411,E2 -4700.411} C_VEL
LIN {X 0,Y 523.904,Z 285.227,A -85,B 0,C 180,E1 -4702.894,E2 -4702.894} C_VEL
LIN {X 0,Y 523.943,Z 285.22,A -85,B 0,C 180,E1 -4705.419,E2 -4705.419} C_VEL
LIN {X 0,Y 523.959,Z 285.21,A -85,B 0,C 180,E1 -4708,E2 -4708} C_VEL
LIN {X 0,Y 523.942,Z 285.219,A -85,B 0,C 180,E1 -4710.857,E2 -4710.857} C_VEL
LIN {X 0,Y 523.952,Z 285.218,A -85,B 0,C 180,E1 -4713.736,E2 -4713.736} C_VEL
LIN {X 0,Y 523.913,Z 285.218,A -85,B 0,C 180,E1 -4716.406,E2 -4716.406} C_VEL
LIN {X 0,Y 523.951,Z 285.219,A -85,B 0,C 180,E1 -4719.082,E2 -4719.082} C_VEL
LIN {X 0,Y 523.949,Z 285.215,A -85,B 0,C 180,E1 -4722.12,E2 -4722.12} C_VEL
LIN {X 0,Y 523.948,Z 285.219,A -85,B 0,C 180,E1 -4725.31,E2 -4725.31} C_VEL
LIN {X 0,Y 523.966,Z 285.213,A -85,B 0,C 180,E1 -4728.689,E2 -4728.689} C_VEL
LIN {X 0,Y 523.919,Z 285.219,A -85,B 0,C 180,E1 -4731.081,E2 -4731.081} C_VEL
LIN {X 0,Y 523.92,Z 285.225,A -85,B 0,C 180,E1 -4733.829,E2 -4733.829} C_VEL
LIN {X 0,Y 523.937,Z 285.217,A -85,B 0,C 180,E1 -4736.637,E2 -4736.637} C_VEL
LIN {X 0,Y 523.952,Z 285.216,A -85,B 0,C 180,E1 -4739.357,E2 -4739.357} C_VEL
LIN {X 0,Y 523.976,Z 285.219,A -85,B 0,C 180,E1 -4742.282,E2 -4742.282} C_VEL
LIN {X 0,Y 523.954,Z 285.222,A -85,B 0,C 180,E1 -4744.583,E2 -4744.583} C_VEL
LIN {X 0,Y 524.013,Z 285.354,A -85,B 0,C 180,E1 -4745.51,E2 -4745.51} C_VEL
LIN {X 0,Y 525.408,Z 294.214,A -85,B 0,C 180,E1 -4746.969,E2 -4746.969} C_VEL
LIN {X 0,Y 524.931,Z 314.059,A -85,B 0,C 180,E1 -4750.039,E2 -4750.039} C_VEL
LIN {X 0,Y 524.503,Z 332.515,A -85,B 0,C 180,E1 -4752.857,E2 -4752.857} C_VEL
LIN {X 0,Y 524.273,Z 345.581,A -85,B 0,C 180,E1 -4754.836,E2 -4754.836} C_VEL
LIN {X 0,Y 525.927,Z 356.7,A -85,B 0,C 180,E1 -4755.043,E2 -4755.043} C_VEL
LIN {X 0,Y 525.465,Z 453.91,A -85,B 0,C 180,E1 -4756.391,E2 -4756.391} C_VEL
LIN {X 0,Y 525.305,Z 467.235,A -85,B 0,C 180,E1 -4756.732,E2 -4756.732} C_VEL
LIN {X 0,Y 525.03,Z 479.432,A -85,B 0,C 180,E1 -4757.192,E2 -4757.192} C_VEL
LIN {X 0,Y 524.865,Z 490.251,A -85,B 0,C 180,E1 -4757.74,E2 -4757.74} C_VEL
LIN {X 0,Y 524.587,Z 500.754,A -85,B 0,C 180,E1 -4758.408,E2 -4758.408} C_VEL
LIN {X 0,Y 524.293,Z 511.689,A -85,B 0,C 180,E1 -4759.282,E2 -4759.282} C_VEL
LIN {X 0,Y 524.041,Z 520.607,A -85,B 0,C 180,E1 -4760.156,E2 -4760.156} C_VEL
LIN {X 0,Y 523.772,Z 530.298,A -85,B 0,C 180,E1 -4761.319,E2 -4761.319} C_VEL
LIN {X 0,Y 523.605,Z 538.014,A -85,B 0,C 180,E1 -4762.482,E2 -4762.482} C_VEL
LIN {X 0,Y 523.482,Z 545.128,A -85,B 0,C 180,E1 -4763.836,E2 -4763.836} C_VEL
LIN {X 0,Y 523.383,Z 549.859,A -85,B 0,C 180,E1 -4764.994,E2 -4764.994} C_VEL
LIN {X 0,Y 523.443,Z 553.479,A -85,B 0,C 180,E1 -4766.152,E2 -4766.152} C_VEL
LIN {X 0,Y 523.367,Z 555.342,A -85,B 0,C 180,E1 -4766.922,E2 -4766.922} C_VEL
LIN {X 0,Y 523.334,Z 556.74,A -85,B 0,C 180,E1 -4767.692,E2 -4767.692} C_VEL
LIN {X 0,Y 523.25,Z 558.344,A -85,B 0,C 180,E1 -4769.232,E2 -4769.232} C_VEL
LIN {X 0,Y 523.25,Z 558.561,A -85,B 0,C 180,E1 -4770.001,E2 -4770.001} C_VEL
LIN {X 0,Y 523.274,Z 557.738,A -85,B 0,C 180,E1 -4771.54,E2 -4771.54} C_VEL
LIN {X 0,Y 523.334,Z 556.743,A -85,B 0,C 180,E1 -4772.31,E2 -4772.31} C_VEL
